(* Logix 5000 project; controller QW361 vendor 1 type 14 code 107 rev 32.11; software revision 32.00; part 14 of 20 *)

        [1996].log_data[0].time := 300.0, [1996].log_data[0].minminute := 50, [1996].log_data[0].maxminute := 50, [1996].log_data[0].valid := 1, [1996].log_data[1].valid := 1, [1996].log_data[2].valid := 1, [1996].log_data[3].valid := 1, [1996].log_data[4].valid := 1, [1996].time.Year := 2022, [1996].time.Month := 4, [1996].time.Day := 30, [1996].time.Hour := 19, [1996].time.Minute := 54, [1996].time.Second := 59, [1996].time.DST_ON := 1, [1997].log_data[0].min := 1.0, [1997].log_data[0].max := 1.0, [1997].log_data[0].total := 300.0, [1997].log_data[0].time := 300.0, [1997].log_data[0].minminute := 55, [1997].log_data[0].maxminute := 55, [1997].log_data[0].valid := 1, [1997].log_data[1].valid := 1, [1997].log_data[2].valid := 1, [1997].log_data[3].valid := 1, [1997].log_data[4].valid := 1, [1997].time.Year := 2022, [1997].time.Month := 4, [1997].time.Day := 30, [1997].time.Hour := 19, [1997].time.Minute := 59, [1997].time.Second := 59, [1997].time.DST_ON := 1, [1998].log_data[0].min := 1.0, [1998].log_data[0].max := 1.0, [1998].log_data[0].total := 300.0, [1998].log_data[0].time := 300.0, [1998].log_data[0].valid := 1, [1998].log_data[1].valid := 1, [1998].log_data[2].valid := 1, [1998].log_data[3].valid := 1, [1998].log_data[4].valid := 1, [1998].time.Year := 2022, [1998].time.Month := 4, [1998].time.Day := 30, [1998].time.Hour := 20, [1998].time.Minute := 4, [1998].time.Second := 59, [1998].time.DST_ON := 1, [1999].log_data[0].min := 1.0, [1999].log_data[0].max := 1.0, [1999].log_data[0].total := 300.0, [1999].log_data[0].time := 300.0, [1999].log_data[0].minminute := 5, [1999].log_data[0].maxminute := 5, [1999].log_data[0].valid := 1, [1999].log_data[1].valid := 1, [1999].log_data[2].valid := 1, [1999].log_data[3].valid := 1, [1999].log_data[4].valid := 1,
        [1999].time.Year := 2022, [1999].time.Month := 4, [1999].time.Day := 30, [1999].time.Hour := 20, [1999].time.Minute := 9, [1999].time.Second := 59, [1999].time.DST_ON := 1, [2000].log_data[0].min := 1.0, [2000].log_data[0].max := 1.0, [2000].log_data[0].total := 300.0, [2000].log_data[0].time := 300.0, [2000].log_data[0].minminute := 10, [2000].log_data[0].maxminute := 10, [2000].log_data[0].valid := 1, [2000].log_data[1].valid := 1, [2000].log_data[2].valid := 1, [2000].log_data[3].valid := 1, [2000].log_data[4].valid := 1, [2000].time.Year := 2022, [2000].time.Month := 4, [2000].time.Day := 30, [2000].time.Hour := 20, [2000].time.Minute := 14, [2000].time.Second := 59, [2000].time.DST_ON := 1, [2001].log_data[0].min := 1.0, [2001].log_data[0].max := 1.0, [2001].log_data[0].total := 300.0, [2001].log_data[0].time := 300.0, [2001].log_data[0].minminute := 15, [2001].log_data[0].maxminute := 15, [2001].log_data[0].valid := 1, [2001].log_data[1].valid := 1, [2001].log_data[2].valid := 1, [2001].log_data[3].valid := 1, [2001].log_data[4].valid := 1, [2001].time.Year := 2022, [2001].time.Month := 4, [2001].time.Day := 30, [2001].time.Hour := 20, [2001].time.Minute := 19, [2001].time.Second := 59, [2001].time.DST_ON := 1, [2002].log_data[0].min := 1.0, [2002].log_data[0].max := 1.0, [2002].log_data[0].total := 300.0, [2002].log_data[0].time := 300.0, [2002].log_data[0].minminute := 20, [2002].log_data[0].maxminute := 20, [2002].log_data[0].valid := 1, [2002].log_data[1].valid := 1, [2002].log_data[2].valid := 1, [2002].log_data[3].valid := 1, [2002].log_data[4].valid := 1, [2002].time.Year := 2022, [2002].time.Month := 4, [2002].time.Day := 30, [2002].time.Hour := 20, [2002].time.Minute := 24, [2002].time.Second := 59,
        [2002].time.DST_ON := 1, [2003].log_data[0].min := 1.0, [2003].log_data[0].max := 1.0, [2003].log_data[0].total := 300.0, [2003].log_data[0].time := 300.0, [2003].log_data[0].minminute := 25, [2003].log_data[0].maxminute := 25, [2003].log_data[0].valid := 1, [2003].log_data[1].valid := 1, [2003].log_data[2].valid := 1, [2003].log_data[3].valid := 1, [2003].log_data[4].valid := 1, [2003].time.Year := 2022, [2003].time.Month := 4, [2003].time.Day := 30, [2003].time.Hour := 20, [2003].time.Minute := 29, [2003].time.Second := 59, [2003].time.DST_ON := 1, [2004].log_data[0].min := 1.0, [2004].log_data[0].max := 1.0, [2004].log_data[0].total := 300.0, [2004].log_data[0].time := 300.0, [2004].log_data[0].minminute := 30, [2004].log_data[0].maxminute := 30, [2004].log_data[0].valid := 1, [2004].log_data[1].valid := 1, [2004].log_data[2].valid := 1, [2004].log_data[3].valid := 1, [2004].log_data[4].valid := 1, [2004].time.Year := 2022, [2004].time.Month := 4, [2004].time.Day := 30, [2004].time.Hour := 20, [2004].time.Minute := 34, [2004].time.Second := 59, [2004].time.DST_ON := 1, [2005].log_data[0].min := 1.0, [2005].log_data[0].max := 1.0, [2005].log_data[0].total := 300.0, [2005].log_data[0].time := 300.0, [2005].log_data[0].minminute := 35, [2005].log_data[0].maxminute := 35, [2005].log_data[0].valid := 1, [2005].log_data[1].valid := 1, [2005].log_data[2].valid := 1, [2005].log_data[3].valid := 1, [2005].log_data[4].valid := 1, [2005].time.Year := 2022, [2005].time.Month := 4, [2005].time.Day := 30, [2005].time.Hour := 20, [2005].time.Minute := 39, [2005].time.Second := 59, [2005].time.DST_ON := 1, [2006].log_data[0].min := 1.0, [2006].log_data[0].max := 1.0, [2006].log_data[0].total := 300.0, [2006].log_data[0].time := 300.0, [2006].log_data[0].minminute := 40,
        [2006].log_data[0].maxminute := 40, [2006].log_data[0].valid := 1, [2006].log_data[1].valid := 1, [2006].log_data[2].valid := 1, [2006].log_data[3].valid := 1, [2006].log_data[4].valid := 1, [2006].time.Year := 2022, [2006].time.Month := 4, [2006].time.Day := 30, [2006].time.Hour := 20, [2006].time.Minute := 44, [2006].time.Second := 59, [2006].time.DST_ON := 1, [2007].log_data[0].min := 1.0, [2007].log_data[0].max := 1.0, [2007].log_data[0].total := 300.0, [2007].log_data[0].time := 300.0, [2007].log_data[0].minminute := 45, [2007].log_data[0].maxminute := 45, [2007].log_data[0].valid := 1, [2007].log_data[1].valid := 1, [2007].log_data[2].valid := 1, [2007].log_data[3].valid := 1, [2007].log_data[4].valid := 1, [2007].time.Year := 2022, [2007].time.Month := 4, [2007].time.Day := 30, [2007].time.Hour := 20, [2007].time.Minute := 49, [2007].time.Second := 59, [2007].time.DST_ON := 1, [2008].log_data[0].min := 1.0, [2008].log_data[0].max := 1.0, [2008].log_data[0].total := 300.001, [2008].log_data[0].time := 300.001, [2008].log_data[0].minminute := 50, [2008].log_data[0].maxminute := 50, [2008].log_data[0].valid := 1, [2008].log_data[1].valid := 1, [2008].log_data[2].valid := 1, [2008].log_data[3].valid := 1, [2008].log_data[4].valid := 1, [2008].time.Year := 2022, [2008].time.Month := 4, [2008].time.Day := 30, [2008].time.Hour := 20, [2008].time.Minute := 54, [2008].time.Second := 59, [2008].time.DST_ON := 1, [2009].log_data[0].min := 1.0, [2009].log_data[0].max := 1.0, [2009].log_data[0].total := 300.001, [2009].log_data[0].time := 300.001, [2009].log_data[0].minminute := 55, [2009].log_data[0].maxminute := 55, [2009].log_data[0].valid := 1, [2009].log_data[1].valid := 1, [2009].log_data[2].valid := 1, [2009].log_data[3].valid := 1, [2009].log_data[4].valid := 1,
        [2009].time.Year := 2022, [2009].time.Month := 4, [2009].time.Day := 30, [2009].time.Hour := 20, [2009].time.Minute := 59, [2009].time.Second := 59, [2009].time.DST_ON := 1, [2010].log_data[0].min := 1.0, [2010].log_data[0].max := 1.0, [2010].log_data[0].total := 300.0, [2010].log_data[0].time := 300.0, [2010].log_data[0].valid := 1, [2010].log_data[1].valid := 1, [2010].log_data[2].valid := 1, [2010].log_data[3].valid := 1, [2010].log_data[4].valid := 1, [2010].time.Year := 2022, [2010].time.Month := 4, [2010].time.Day := 30, [2010].time.Hour := 21, [2010].time.Minute := 4, [2010].time.Second := 59, [2010].time.DST_ON := 1, [2011].log_data[0].min := 1.0, [2011].log_data[0].max := 1.0, [2011].log_data[0].total := 300.0, [2011].log_data[0].time := 300.0, [2011].log_data[0].minminute := 5, [2011].log_data[0].maxminute := 5, [2011].log_data[0].valid := 1, [2011].log_data[1].valid := 1, [2011].log_data[2].valid := 1, [2011].log_data[3].valid := 1, [2011].log_data[4].valid := 1, [2011].time.Year := 2022, [2011].time.Month := 4, [2011].time.Day := 30, [2011].time.Hour := 21, [2011].time.Minute := 9, [2011].time.Second := 59, [2011].time.DST_ON := 1, [2012].log_data[0].min := 1.0, [2012].log_data[0].max := 1.0, [2012].log_data[0].total := 300.0, [2012].log_data[0].time := 300.0, [2012].log_data[0].minminute := 10, [2012].log_data[0].maxminute := 10, [2012].log_data[0].valid := 1, [2012].log_data[1].valid := 1, [2012].log_data[2].valid := 1, [2012].log_data[3].valid := 1, [2012].log_data[4].valid := 1, [2012].time.Year := 2022, [2012].time.Month := 4, [2012].time.Day := 30, [2012].time.Hour := 21, [2012].time.Minute := 14, [2012].time.Second := 59, [2012].time.DST_ON := 1, [2013].log_data[0].min := 1.0,
        [2013].log_data[0].max := 1.0, [2013].log_data[0].total := 300.0, [2013].log_data[0].time := 300.0, [2013].log_data[0].minminute := 15, [2013].log_data[0].maxminute := 15, [2013].log_data[0].valid := 1, [2013].log_data[1].valid := 1, [2013].log_data[2].valid := 1, [2013].log_data[3].valid := 1, [2013].log_data[4].valid := 1, [2013].time.Year := 2022, [2013].time.Month := 4, [2013].time.Day := 30, [2013].time.Hour := 21, [2013].time.Minute := 19, [2013].time.Second := 59, [2013].time.DST_ON := 1, [2014].log_data[0].min := 1.0, [2014].log_data[0].max := 1.0, [2014].log_data[0].total := 300.0, [2014].log_data[0].time := 300.0, [2014].log_data[0].minminute := 20, [2014].log_data[0].maxminute := 20, [2014].log_data[0].valid := 1, [2014].log_data[1].valid := 1, [2014].log_data[2].valid := 1, [2014].log_data[3].valid := 1, [2014].log_data[4].valid := 1, [2014].time.Year := 2022, [2014].time.Month := 4, [2014].time.Day := 30, [2014].time.Hour := 21, [2014].time.Minute := 24, [2014].time.Second := 59, [2014].time.DST_ON := 1, [2015].log_data[0].min := 1.0, [2015].log_data[0].max := 1.0, [2015].log_data[0].total := 300.0, [2015].log_data[0].time := 300.0, [2015].log_data[0].minminute := 25, [2015].log_data[0].maxminute := 25, [2015].log_data[0].valid := 1, [2015].log_data[1].valid := 1, [2015].log_data[2].valid := 1, [2015].log_data[3].valid := 1, [2015].log_data[4].valid := 1, [2015].time.Year := 2022, [2015].time.Month := 4, [2015].time.Day := 30, [2015].time.Hour := 21, [2015].time.Minute := 29, [2015].time.Second := 59, [2015].time.DST_ON := 1, [2016].log_data[0].min := 1.0, [2016].log_data[0].max := 1.0, [2016].log_data[0].total := 300.0, [2016].log_data[0].time := 300.0, [2016].log_data[0].minminute := 30, [2016].log_data[0].maxminute := 30, [2016].log_data[0].valid := 1,
        [2016].log_data[1].valid := 1, [2016].log_data[2].valid := 1, [2016].log_data[3].valid := 1, [2016].log_data[4].valid := 1, [2016].time.Year := 2022, [2016].time.Month := 4, [2016].time.Day := 30, [2016].time.Hour := 21, [2016].time.Minute := 34, [2016].time.Second := 59, [2016].time.DST_ON := 1, [2017].log_data[0].min := 1.0, [2017].log_data[0].max := 1.0, [2017].log_data[0].total := 300.0, [2017].log_data[0].time := 300.0, [2017].log_data[0].minminute := 35, [2017].log_data[0].maxminute := 35, [2017].log_data[0].valid := 1, [2017].log_data[1].valid := 1, [2017].log_data[2].valid := 1, [2017].log_data[3].valid := 1, [2017].log_data[4].valid := 1, [2017].time.Year := 2022, [2017].time.Month := 4, [2017].time.Day := 30, [2017].time.Hour := 21, [2017].time.Minute := 39, [2017].time.Second := 59, [2017].time.DST_ON := 1, [2018].log_data[0].min := 1.0, [2018].log_data[0].max := 1.0, [2018].log_data[0].total := 300.0, [2018].log_data[0].time := 300.0, [2018].log_data[0].minminute := 40, [2018].log_data[0].maxminute := 40, [2018].log_data[0].valid := 1, [2018].log_data[1].valid := 1, [2018].log_data[2].valid := 1, [2018].log_data[3].valid := 1, [2018].log_data[4].valid := 1, [2018].time.Year := 2022, [2018].time.Month := 4, [2018].time.Day := 30, [2018].time.Hour := 21, [2018].time.Minute := 44, [2018].time.Second := 59, [2018].time.DST_ON := 1, [2019].log_data[0].min := 1.0, [2019].log_data[0].max := 1.0, [2019].log_data[0].total := 300.0, [2019].log_data[0].time := 300.0, [2019].log_data[0].minminute := 45, [2019].log_data[0].maxminute := 45, [2019].log_data[0].valid := 1, [2019].log_data[1].valid := 1, [2019].log_data[2].valid := 1, [2019].log_data[3].valid := 1, [2019].log_data[4].valid := 1, [2019].time.Year := 2022, [2019].time.Month := 4,
        [2019].time.Day := 30, [2019].time.Hour := 21, [2019].time.Minute := 49, [2019].time.Second := 59, [2019].time.DST_ON := 1, [2020].log_data[0].min := 1.0, [2020].log_data[0].max := 1.0, [2020].log_data[0].total := 300.0, [2020].log_data[0].time := 300.0, [2020].log_data[0].minminute := 50, [2020].log_data[0].maxminute := 50, [2020].log_data[0].valid := 1, [2020].log_data[1].valid := 1, [2020].log_data[2].valid := 1, [2020].log_data[3].valid := 1, [2020].log_data[4].valid := 1, [2020].time.Year := 2022, [2020].time.Month := 4, [2020].time.Day := 30, [2020].time.Hour := 21, [2020].time.Minute := 54, [2020].time.Second := 59, [2020].time.DST_ON := 1, [2021].log_data[0].min := 1.0, [2021].log_data[0].max := 1.0, [2021].log_data[0].total := 300.0, [2021].log_data[0].time := 300.0, [2021].log_data[0].minminute := 55, [2021].log_data[0].maxminute := 55, [2021].log_data[0].valid := 1, [2021].log_data[1].valid := 1, [2021].log_data[2].valid := 1, [2021].log_data[3].valid := 1, [2021].log_data[4].valid := 1, [2021].time.Year := 2022, [2021].time.Month := 4, [2021].time.Day := 30, [2021].time.Hour := 21, [2021].time.Minute := 59, [2021].time.Second := 59, [2021].time.DST_ON := 1, [2022].log_data[0].min := 1.0, [2022].log_data[0].max := 1.0, [2022].log_data[0].total := 300.0, [2022].log_data[0].time := 300.0, [2022].log_data[0].valid := 1, [2022].log_data[1].valid := 1, [2022].log_data[2].valid := 1, [2022].log_data[3].valid := 1, [2022].log_data[4].valid := 1, [2022].time.Year := 2022, [2022].time.Month := 4, [2022].time.Day := 30, [2022].time.Hour := 22, [2022].time.Minute := 4, [2022].time.Second := 59, [2022].time.DST_ON := 1, [2023].log_data[0].min := 1.0, [2023].log_data[0].max := 1.0, [2023].log_data[0].total := 300.0,
        [2023].log_data[0].time := 300.0, [2023].log_data[0].minminute := 5, [2023].log_data[0].maxminute := 5, [2023].log_data[0].valid := 1, [2023].log_data[1].valid := 1, [2023].log_data[2].valid := 1, [2023].log_data[3].valid := 1, [2023].log_data[4].valid := 1, [2023].time.Year := 2022, [2023].time.Month := 4, [2023].time.Day := 30, [2023].time.Hour := 22, [2023].time.Minute := 9, [2023].time.Second := 59, [2023].time.DST_ON := 1, [2024].log_data[0].min := 1.0, [2024].log_data[0].max := 1.0, [2024].log_data[0].total := 300.0, [2024].log_data[0].time := 300.0, [2024].log_data[0].minminute := 10, [2024].log_data[0].maxminute := 10, [2024].log_data[0].valid := 1, [2024].log_data[1].valid := 1, [2024].log_data[2].valid := 1, [2024].log_data[3].valid := 1, [2024].log_data[4].valid := 1, [2024].time.Year := 2022, [2024].time.Month := 4, [2024].time.Day := 30, [2024].time.Hour := 22, [2024].time.Minute := 14, [2024].time.Second := 59, [2024].time.DST_ON := 1, [2025].log_data[0].min := 1.0, [2025].log_data[0].max := 1.0, [2025].log_data[0].total := 300.0, [2025].log_data[0].time := 300.0, [2025].log_data[0].minminute := 15, [2025].log_data[0].maxminute := 15, [2025].log_data[0].valid := 1, [2025].log_data[1].valid := 1, [2025].log_data[2].valid := 1, [2025].log_data[3].valid := 1, [2025].log_data[4].valid := 1, [2025].time.Year := 2022, [2025].time.Month := 4, [2025].time.Day := 30, [2025].time.Hour := 22, [2025].time.Minute := 19, [2025].time.Second := 59, [2025].time.DST_ON := 1, [2026].log_data[0].min := 1.0, [2026].log_data[0].max := 1.0, [2026].log_data[0].total := 300.0, [2026].log_data[0].time := 300.0, [2026].log_data[0].minminute := 20, [2026].log_data[0].maxminute := 20, [2026].log_data[0].valid := 1, [2026].log_data[1].valid := 1, [2026].log_data[2].valid := 1,
        [2026].log_data[3].valid := 1, [2026].log_data[4].valid := 1, [2026].time.Year := 2022, [2026].time.Month := 4, [2026].time.Day := 30, [2026].time.Hour := 22, [2026].time.Minute := 24, [2026].time.Second := 59, [2026].time.DST_ON := 1, [2027].log_data[0].min := 1.0, [2027].log_data[0].max := 1.0, [2027].log_data[0].total := 300.0, [2027].log_data[0].time := 300.0, [2027].log_data[0].minminute := 25, [2027].log_data[0].maxminute := 25, [2027].log_data[0].valid := 1, [2027].log_data[1].valid := 1, [2027].log_data[2].valid := 1, [2027].log_data[3].valid := 1, [2027].log_data[4].valid := 1, [2027].time.Year := 2022, [2027].time.Month := 4, [2027].time.Day := 30, [2027].time.Hour := 22, [2027].time.Minute := 29, [2027].time.Second := 59, [2027].time.DST_ON := 1, [2028].log_data[0].min := 1.0, [2028].log_data[0].max := 1.0, [2028].log_data[0].total := 300.0, [2028].log_data[0].time := 300.0, [2028].log_data[0].minminute := 30, [2028].log_data[0].maxminute := 30, [2028].log_data[0].valid := 1, [2028].log_data[1].valid := 1, [2028].log_data[2].valid := 1, [2028].log_data[3].valid := 1, [2028].log_data[4].valid := 1, [2028].time.Year := 2022, [2028].time.Month := 4, [2028].time.Day := 30, [2028].time.Hour := 22, [2028].time.Minute := 34, [2028].time.Second := 59, [2028].time.DST_ON := 1, [2029].log_data[0].min := 1.0, [2029].log_data[0].max := 1.0, [2029].log_data[0].total := 300.0, [2029].log_data[0].time := 300.0, [2029].log_data[0].minminute := 35, [2029].log_data[0].maxminute := 35, [2029].log_data[0].valid := 1, [2029].log_data[1].valid := 1, [2029].log_data[2].valid := 1, [2029].log_data[3].valid := 1, [2029].log_data[4].valid := 1, [2029].time.Year := 2022, [2029].time.Month := 4, [2029].time.Day := 30, [2029].time.Hour := 22,
        [2029].time.Minute := 39, [2029].time.Second := 59, [2029].time.DST_ON := 1, [2030].log_data[0].min := 1.0, [2030].log_data[0].max := 1.0, [2030].log_data[0].total := 300.0, [2030].log_data[0].time := 300.0, [2030].log_data[0].minminute := 40, [2030].log_data[0].maxminute := 40, [2030].log_data[0].valid := 1, [2030].log_data[1].valid := 1, [2030].log_data[2].valid := 1, [2030].log_data[3].valid := 1, [2030].log_data[4].valid := 1, [2030].time.Year := 2022, [2030].time.Month := 4, [2030].time.Day := 30, [2030].time.Hour := 22, [2030].time.Minute := 44, [2030].time.Second := 59, [2030].time.DST_ON := 1, [2031].log_data[0].min := 1.0, [2031].log_data[0].max := 1.0, [2031].log_data[0].total := 300.0, [2031].log_data[0].time := 300.0, [2031].log_data[0].minminute := 45, [2031].log_data[0].maxminute := 45, [2031].log_data[0].valid := 1, [2031].log_data[1].valid := 1, [2031].log_data[2].valid := 1, [2031].log_data[3].valid := 1, [2031].log_data[4].valid := 1, [2031].time.Year := 2022, [2031].time.Month := 4, [2031].time.Day := 30, [2031].time.Hour := 22, [2031].time.Minute := 49, [2031].time.Second := 59, [2031].time.DST_ON := 1, [2032].log_data[0].min := 1.0, [2032].log_data[0].max := 1.0, [2032].log_data[0].total := 300.0, [2032].log_data[0].time := 300.0, [2032].log_data[0].minminute := 50, [2032].log_data[0].maxminute := 50, [2032].log_data[0].valid := 1, [2032].log_data[1].valid := 1, [2032].log_data[2].valid := 1, [2032].log_data[3].valid := 1, [2032].log_data[4].valid := 1, [2032].time.Year := 2022, [2032].time.Month := 4, [2032].time.Day := 30, [2032].time.Hour := 22, [2032].time.Minute := 54, [2032].time.Second := 59, [2032].time.DST_ON := 1, [2033].log_data[0].min := 1.0, [2033].log_data[0].max := 1.0, [2033].log_data[0].total := 300.0,
        [2033].log_data[0].time := 300.0, [2033].log_data[0].minminute := 55, [2033].log_data[0].maxminute := 55, [2033].log_data[0].valid := 1, [2033].log_data[1].valid := 1, [2033].log_data[2].valid := 1, [2033].log_data[3].valid := 1, [2033].log_data[4].valid := 1, [2033].time.Year := 2022, [2033].time.Month := 4, [2033].time.Day := 30, [2033].time.Hour := 22, [2033].time.Minute := 59, [2033].time.Second := 59, [2033].time.DST_ON := 1, [2034].log_data[0].min := 1.0, [2034].log_data[0].max := 1.0, [2034].log_data[0].total := 300.0, [2034].log_data[0].time := 300.0, [2034].log_data[0].valid := 1, [2034].log_data[1].valid := 1, [2034].log_data[2].valid := 1, [2034].log_data[3].valid := 1, [2034].log_data[4].valid := 1, [2034].time.Year := 2022, [2034].time.Month := 4, [2034].time.Day := 30, [2034].time.Hour := 23, [2034].time.Minute := 4, [2034].time.Second := 59, [2034].time.DST_ON := 1, [2035].log_data[0].min := 1.0, [2035].log_data[0].max := 1.0, [2035].log_data[0].total := 300.0, [2035].log_data[0].time := 300.0, [2035].log_data[0].minminute := 5, [2035].log_data[0].maxminute := 5, [2035].log_data[0].valid := 1, [2035].log_data[1].valid := 1, [2035].log_data[2].valid := 1, [2035].log_data[3].valid := 1, [2035].log_data[4].valid := 1, [2035].time.Year := 2022, [2035].time.Month := 4, [2035].time.Day := 30, [2035].time.Hour := 23, [2035].time.Minute := 9, [2035].time.Second := 59, [2035].time.DST_ON := 1, [2036].log_data[0].min := 1.0, [2036].log_data[0].max := 1.0, [2036].log_data[0].total := 300.0, [2036].log_data[0].time := 300.0, [2036].log_data[0].minminute := 10, [2036].log_data[0].maxminute := 10, [2036].log_data[0].valid := 1, [2036].log_data[1].valid := 1, [2036].log_data[2].valid := 1, [2036].log_data[3].valid := 1, [2036].log_data[4].valid := 1,
        [2036].time.Year := 2022, [2036].time.Month := 4, [2036].time.Day := 30, [2036].time.Hour := 23, [2036].time.Minute := 14, [2036].time.Second := 59, [2036].time.DST_ON := 1, [2037].log_data[0].min := 1.0, [2037].log_data[0].max := 1.0, [2037].log_data[0].total := 300.0, [2037].log_data[0].time := 300.0, [2037].log_data[0].minminute := 15, [2037].log_data[0].maxminute := 15, [2037].log_data[0].valid := 1, [2037].log_data[1].valid := 1, [2037].log_data[2].valid := 1, [2037].log_data[3].valid := 1, [2037].log_data[4].valid := 1, [2037].time.Year := 2022, [2037].time.Month := 4, [2037].time.Day := 30, [2037].time.Hour := 23, [2037].time.Minute := 19, [2037].time.Second := 59, [2037].time.DST_ON := 1, [2038].log_data[0].min := 1.0, [2038].log_data[0].max := 1.0, [2038].log_data[0].total := 300.0, [2038].log_data[0].time := 300.0, [2038].log_data[0].minminute := 20, [2038].log_data[0].maxminute := 20, [2038].log_data[0].valid := 1, [2038].log_data[1].valid := 1, [2038].log_data[2].valid := 1, [2038].log_data[3].valid := 1, [2038].log_data[4].valid := 1, [2038].time.Year := 2022, [2038].time.Month := 4, [2038].time.Day := 30, [2038].time.Hour := 23, [2038].time.Minute := 24, [2038].time.Second := 59, [2038].time.DST_ON := 1, [2039].log_data[0].min := 1.0, [2039].log_data[0].max := 1.0, [2039].log_data[0].total := 300.0, [2039].log_data[0].time := 300.0, [2039].log_data[0].minminute := 25, [2039].log_data[0].maxminute := 25, [2039].log_data[0].valid := 1, [2039].log_data[1].valid := 1, [2039].log_data[2].valid := 1, [2039].log_data[3].valid := 1, [2039].log_data[4].valid := 1, [2039].time.Year := 2022, [2039].time.Month := 4, [2039].time.Day := 30, [2039].time.Hour := 23, [2039].time.Minute := 29, [2039].time.Second := 59,
        [2039].time.DST_ON := 1, [2040].log_data[0].min := 1.0, [2040].log_data[0].max := 1.0, [2040].log_data[0].total := 300.0, [2040].log_data[0].time := 300.0, [2040].log_data[0].minminute := 30, [2040].log_data[0].maxminute := 30, [2040].log_data[0].valid := 1, [2040].log_data[1].valid := 1, [2040].log_data[2].valid := 1, [2040].log_data[3].valid := 1, [2040].log_data[4].valid := 1, [2040].time.Year := 2022, [2040].time.Month := 4, [2040].time.Day := 30, [2040].time.Hour := 23, [2040].time.Minute := 34, [2040].time.Second := 59, [2040].time.DST_ON := 1, [2041].log_data[0].min := 1.0, [2041].log_data[0].max := 1.0, [2041].log_data[0].total := 300.0, [2041].log_data[0].time := 300.0, [2041].log_data[0].minminute := 35, [2041].log_data[0].maxminute := 35, [2041].log_data[0].valid := 1, [2041].log_data[1].valid := 1, [2041].log_data[2].valid := 1, [2041].log_data[3].valid := 1, [2041].log_data[4].valid := 1, [2041].time.Year := 2022, [2041].time.Month := 4, [2041].time.Day := 30, [2041].time.Hour := 23, [2041].time.Minute := 39, [2041].time.Second := 59, [2041].time.DST_ON := 1, [2042].log_data[0].min := 1.0, [2042].log_data[0].max := 1.0, [2042].log_data[0].total := 300.0, [2042].log_data[0].time := 300.0, [2042].log_data[0].minminute := 40, [2042].log_data[0].maxminute := 40, [2042].log_data[0].valid := 1, [2042].log_data[1].valid := 1, [2042].log_data[2].valid := 1, [2042].log_data[3].valid := 1, [2042].log_data[4].valid := 1, [2042].time.Year := 2022, [2042].time.Month := 4, [2042].time.Day := 30, [2042].time.Hour := 23, [2042].time.Minute := 44, [2042].time.Second := 59, [2042].time.DST_ON := 1, [2043].log_data[0].min := 1.0, [2043].log_data[0].max := 1.0, [2043].log_data[0].total := 300.0, [2043].log_data[0].time := 300.0, [2043].log_data[0].minminute := 45,
        [2043].log_data[0].maxminute := 45, [2043].log_data[0].valid := 1, [2043].log_data[1].valid := 1, [2043].log_data[2].valid := 1, [2043].log_data[3].valid := 1, [2043].log_data[4].valid := 1, [2043].time.Year := 2022, [2043].time.Month := 4, [2043].time.Day := 30, [2043].time.Hour := 23, [2043].time.Minute := 49, [2043].time.Second := 59, [2043].time.DST_ON := 1, [2044].log_data[0].min := 1.0, [2044].log_data[0].max := 1.0, [2044].log_data[0].total := 300.0, [2044].log_data[0].time := 300.0, [2044].log_data[0].minminute := 50, [2044].log_data[0].maxminute := 50, [2044].log_data[0].valid := 1, [2044].log_data[1].valid := 1, [2044].log_data[2].valid := 1, [2044].log_data[3].valid := 1, [2044].log_data[4].valid := 1, [2044].time.Year := 2022, [2044].time.Month := 4, [2044].time.Day := 30, [2044].time.Hour := 23, [2044].time.Minute := 54, [2044].time.Second := 59, [2044].time.DST_ON := 1, [2045].log_data[0].min := 1.0, [2045].log_data[0].max := 1.0, [2045].log_data[0].total := 300.0, [2045].log_data[0].time := 300.0, [2045].log_data[0].minminute := 55, [2045].log_data[0].maxminute := 55, [2045].log_data[0].valid := 1, [2045].log_data[1].valid := 1, [2045].log_data[2].valid := 1, [2045].log_data[3].valid := 1, [2045].log_data[4].valid := 1, [2045].time.Year := 2022, [2045].time.Month := 4, [2045].time.Day := 30, [2045].time.Hour := 23, [2045].time.Minute := 59, [2045].time.Second := 59, [2045].time.DST_ON := 1, [2046].log_data[0].min := 1.0, [2046].log_data[0].max := 1.0, [2046].log_data[0].total := 300.0, [2046].log_data[0].time := 300.0, [2046].log_data[0].valid := 1, [2046].log_data[1].valid := 1, [2046].log_data[2].valid := 1, [2046].log_data[3].valid := 1, [2046].log_data[4].valid := 1, [2046].time.Year := 2022, [2046].time.Month := 5,
        [2046].time.Day := 1, [2046].time.Minute := 4, [2046].time.Second := 59, [2046].time.DST_ON := 1, [2047].log_data[0].min := 1.0, [2047].log_data[0].max := 1.0, [2047].log_data[0].total := 300.0, [2047].log_data[0].time := 300.0, [2047].log_data[0].minminute := 5, [2047].log_data[0].maxminute := 5, [2047].log_data[0].valid := 1, [2047].log_data[1].valid := 1, [2047].log_data[2].valid := 1, [2047].log_data[3].valid := 1, [2047].log_data[4].valid := 1, [2047].time.Year := 2022, [2047].time.Month := 5, [2047].time.Day := 1, [2047].time.Minute := 9, [2047].time.Second := 59, [2047].time.DST_ON := 1, [2048].log_data[0].min := 1.0, [2048].log_data[0].max := 1.0, [2048].log_data[0].total := 300.0, [2048].log_data[0].time := 300.0, [2048].log_data[0].minminute := 10, [2048].log_data[0].maxminute := 10, [2048].log_data[0].valid := 1, [2048].log_data[1].valid := 1, [2048].log_data[2].valid := 1, [2048].log_data[3].valid := 1, [2048].log_data[4].valid := 1, [2048].time.Year := 2022, [2048].time.Month := 5, [2048].time.Day := 1, [2048].time.Minute := 14, [2048].time.Second := 59, [2048].time.DST_ON := 1, [2049].log_data[0].min := 1.0, [2049].log_data[0].max := 1.0, [2049].log_data[0].total := 300.0, [2049].log_data[0].time := 300.0, [2049].log_data[0].minminute := 15, [2049].log_data[0].maxminute := 15, [2049].log_data[0].valid := 1, [2049].log_data[1].valid := 1, [2049].log_data[2].valid := 1, [2049].log_data[3].valid := 1, [2049].log_data[4].valid := 1, [2049].time.Year := 2022, [2049].time.Month := 5, [2049].time.Day := 1, [2049].time.Minute := 19, [2049].time.Second := 59, [2049].time.DST_ON := 1, [2050].log_data[0].min := 1.0, [2050].log_data[0].max := 1.0, [2050].log_data[0].total := 300.0, [2050].log_data[0].time := 300.0, [2050].log_data[0].minminute := 20,
        [2050].log_data[0].maxminute := 20, [2050].log_data[0].valid := 1, [2050].log_data[1].valid := 1, [2050].log_data[2].valid := 1, [2050].log_data[3].valid := 1, [2050].log_data[4].valid := 1, [2050].time.Year := 2022, [2050].time.Month := 5, [2050].time.Day := 1, [2050].time.Minute := 24, [2050].time.Second := 59, [2050].time.DST_ON := 1, [2051].log_data[0].min := 1.0, [2051].log_data[0].max := 1.0, [2051].log_data[0].total := 300.0, [2051].log_data[0].time := 300.0, [2051].log_data[0].minminute := 25, [2051].log_data[0].maxminute := 25, [2051].log_data[0].valid := 1, [2051].log_data[1].valid := 1, [2051].log_data[2].valid := 1, [2051].log_data[3].valid := 1, [2051].log_data[4].valid := 1, [2051].time.Year := 2022, [2051].time.Month := 5, [2051].time.Day := 1, [2051].time.Minute := 29, [2051].time.Second := 59, [2051].time.DST_ON := 1, [2052].log_data[0].min := 1.0, [2052].log_data[0].max := 1.0, [2052].log_data[0].total := 300.0, [2052].log_data[0].time := 300.0, [2052].log_data[0].minminute := 30, [2052].log_data[0].maxminute := 30, [2052].log_data[0].valid := 1, [2052].log_data[1].valid := 1, [2052].log_data[2].valid := 1, [2052].log_data[3].valid := 1, [2052].log_data[4].valid := 1, [2052].time.Year := 2022, [2052].time.Month := 5, [2052].time.Day := 1, [2052].time.Minute := 34, [2052].time.Second := 59, [2052].time.DST_ON := 1, [2053].log_data[0].min := 1.0, [2053].log_data[0].max := 1.0, [2053].log_data[0].total := 299.999, [2053].log_data[0].time := 299.999, [2053].log_data[0].minminute := 35, [2053].log_data[0].maxminute := 35, [2053].log_data[0].valid := 1, [2053].log_data[1].valid := 1, [2053].log_data[2].valid := 1, [2053].log_data[3].valid := 1, [2053].log_data[4].valid := 1, [2053].time.Year := 2022, [2053].time.Month := 5, [2053].time.Day := 1,
        [2053].time.Minute := 39, [2053].time.Second := 59, [2053].time.DST_ON := 1, [2054].log_data[0].min := 1.0, [2054].log_data[0].max := 1.0, [2054].log_data[0].total := 300.0, [2054].log_data[0].time := 300.0, [2054].log_data[0].minminute := 40, [2054].log_data[0].maxminute := 40, [2054].log_data[0].valid := 1, [2054].log_data[1].valid := 1, [2054].log_data[2].valid := 1, [2054].log_data[3].valid := 1, [2054].log_data[4].valid := 1, [2054].time.Year := 2022, [2054].time.Month := 5, [2054].time.Day := 1, [2054].time.Minute := 44, [2054].time.Second := 59, [2054].time.DST_ON := 1, [2055].log_data[0].min := 1.0, [2055].log_data[0].max := 1.0, [2055].log_data[0].total := 300.0, [2055].log_data[0].time := 300.0, [2055].log_data[0].minminute := 45, [2055].log_data[0].maxminute := 45, [2055].log_data[0].valid := 1, [2055].log_data[1].valid := 1, [2055].log_data[2].valid := 1, [2055].log_data[3].valid := 1, [2055].log_data[4].valid := 1, [2055].time.Year := 2022, [2055].time.Month := 5, [2055].time.Day := 1, [2055].time.Minute := 49, [2055].time.Second := 59, [2055].time.DST_ON := 1, [2056].log_data[0].min := 1.0, [2056].log_data[0].max := 1.0, [2056].log_data[0].total := 300.0, [2056].log_data[0].time := 300.0, [2056].log_data[0].minminute := 50, [2056].log_data[0].maxminute := 50, [2056].log_data[0].valid := 1, [2056].log_data[1].valid := 1, [2056].log_data[2].valid := 1, [2056].log_data[3].valid := 1, [2056].log_data[4].valid := 1, [2056].time.Year := 2022, [2056].time.Month := 5, [2056].time.Day := 1, [2056].time.Minute := 54, [2056].time.Second := 59, [2056].time.DST_ON := 1, [2057].log_data[0].min := 1.0, [2057].log_data[0].max := 1.0, [2057].log_data[0].total := 300.001, [2057].log_data[0].time := 300.001, [2057].log_data[0].minminute := 55, [2057].log_data[0].maxminute := 55,
        [2057].log_data[0].valid := 1, [2057].log_data[1].valid := 1, [2057].log_data[2].valid := 1, [2057].log_data[3].valid := 1, [2057].log_data[4].valid := 1, [2057].time.Year := 2022, [2057].time.Month := 5, [2057].time.Day := 1, [2057].time.Minute := 59, [2057].time.Second := 59, [2057].time.DST_ON := 1, [2058].log_data[0].min := 1.0, [2058].log_data[0].max := 1.0, [2058].log_data[0].total := 300.0, [2058].log_data[0].time := 300.0, [2058].log_data[0].valid := 1, [2058].log_data[1].valid := 1, [2058].log_data[2].valid := 1, [2058].log_data[3].valid := 1, [2058].log_data[4].valid := 1, [2058].time.Year := 2022, [2058].time.Month := 5, [2058].time.Day := 1, [2058].time.Hour := 1, [2058].time.Minute := 4, [2058].time.Second := 59, [2058].time.DST_ON := 1, [2059].log_data[0].min := 1.0, [2059].log_data[0].max := 1.0, [2059].log_data[0].total := 300.0, [2059].log_data[0].time := 300.0, [2059].log_data[0].minminute := 5, [2059].log_data[0].maxminute := 5, [2059].log_data[0].valid := 1, [2059].log_data[1].valid := 1, [2059].log_data[2].valid := 1, [2059].log_data[3].valid := 1, [2059].log_data[4].valid := 1, [2059].time.Year := 2022, [2059].time.Month := 5, [2059].time.Day := 1, [2059].time.Hour := 1, [2059].time.Minute := 9, [2059].time.Second := 59, [2059].time.DST_ON := 1, [2060].log_data[0].min := 1.0, [2060].log_data[0].max := 1.0, [2060].log_data[0].total := 300.0, [2060].log_data[0].time := 300.0, [2060].log_data[0].minminute := 10, [2060].log_data[0].maxminute := 10, [2060].log_data[0].valid := 1, [2060].log_data[1].valid := 1, [2060].log_data[2].valid := 1, [2060].log_data[3].valid := 1, [2060].log_data[4].valid := 1, [2060].time.Year := 2022, [2060].time.Month := 5, [2060].time.Day := 1, [2060].time.Hour := 1,
        [2060].time.Minute := 14, [2060].time.Second := 59, [2060].time.DST_ON := 1, [2061].log_data[0].min := 1.0, [2061].log_data[0].max := 1.0, [2061].log_data[0].total := 300.0, [2061].log_data[0].time := 300.0, [2061].log_data[0].minminute := 15, [2061].log_data[0].maxminute := 15, [2061].log_data[0].valid := 1, [2061].log_data[1].valid := 1, [2061].log_data[2].valid := 1, [2061].log_data[3].valid := 1, [2061].log_data[4].valid := 1, [2061].time.Year := 2022, [2061].time.Month := 5, [2061].time.Day := 1, [2061].time.Hour := 1, [2061].time.Minute := 19, [2061].time.Second := 59, [2061].time.DST_ON := 1, [2062].log_data[0].min := 1.0, [2062].log_data[0].max := 1.0, [2062].log_data[0].total := 300.0, [2062].log_data[0].time := 300.0, [2062].log_data[0].minminute := 20, [2062].log_data[0].maxminute := 20, [2062].log_data[0].valid := 1, [2062].log_data[1].valid := 1, [2062].log_data[2].valid := 1, [2062].log_data[3].valid := 1, [2062].log_data[4].valid := 1, [2062].time.Year := 2022, [2062].time.Month := 5, [2062].time.Day := 1, [2062].time.Hour := 1, [2062].time.Minute := 24, [2062].time.Second := 59, [2062].time.DST_ON := 1, [2063].log_data[0].min := 1.0, [2063].log_data[0].max := 1.0, [2063].log_data[0].total := 300.0, [2063].log_data[0].time := 300.0, [2063].log_data[0].minminute := 25, [2063].log_data[0].maxminute := 25, [2063].log_data[0].valid := 1, [2063].log_data[1].valid := 1, [2063].log_data[2].valid := 1, [2063].log_data[3].valid := 1, [2063].log_data[4].valid := 1, [2063].time.Year := 2022, [2063].time.Month := 5, [2063].time.Day := 1, [2063].time.Hour := 1, [2063].time.Minute := 29, [2063].time.Second := 59, [2063].time.DST_ON := 1, [2064].log_data[0].min := 1.0, [2064].log_data[0].max := 1.0, [2064].log_data[0].total := 300.0,
        [2064].log_data[0].time := 300.0, [2064].log_data[0].minminute := 30, [2064].log_data[0].maxminute := 30, [2064].log_data[0].valid := 1, [2064].log_data[1].valid := 1, [2064].log_data[2].valid := 1, [2064].log_data[3].valid := 1, [2064].log_data[4].valid := 1, [2064].time.Year := 2022, [2064].time.Month := 5, [2064].time.Day := 1, [2064].time.Hour := 1, [2064].time.Minute := 34, [2064].time.Second := 59, [2064].time.DST_ON := 1, [2065].log_data[0].min := 1.0, [2065].log_data[0].max := 1.0, [2065].log_data[0].total := 300.0, [2065].log_data[0].time := 300.0, [2065].log_data[0].minminute := 35, [2065].log_data[0].maxminute := 35, [2065].log_data[0].valid := 1, [2065].log_data[1].valid := 1, [2065].log_data[2].valid := 1, [2065].log_data[3].valid := 1, [2065].log_data[4].valid := 1, [2065].time.Year := 2022, [2065].time.Month := 5, [2065].time.Day := 1, [2065].time.Hour := 1, [2065].time.Minute := 39, [2065].time.Second := 59, [2065].time.DST_ON := 1, [2066].log_data[0].min := 1.0, [2066].log_data[0].max := 1.0, [2066].log_data[0].total := 300.0, [2066].log_data[0].time := 300.0, [2066].log_data[0].minminute := 40, [2066].log_data[0].maxminute := 40, [2066].log_data[0].valid := 1, [2066].log_data[1].valid := 1, [2066].log_data[2].valid := 1, [2066].log_data[3].valid := 1, [2066].log_data[4].valid := 1, [2066].time.Year := 2022, [2066].time.Month := 5, [2066].time.Day := 1, [2066].time.Hour := 1, [2066].time.Minute := 44, [2066].time.Second := 59, [2066].time.DST_ON := 1, [2067].log_data[0].min := 1.0, [2067].log_data[0].max := 1.0, [2067].log_data[0].total := 300.0, [2067].log_data[0].time := 300.0, [2067].log_data[0].minminute := 45, [2067].log_data[0].maxminute := 45, [2067].log_data[0].valid := 1, [2067].log_data[1].valid := 1, [2067].log_data[2].valid := 1,
        [2067].log_data[3].valid := 1, [2067].log_data[4].valid := 1, [2067].time.Year := 2022, [2067].time.Month := 5, [2067].time.Day := 1, [2067].time.Hour := 1, [2067].time.Minute := 49, [2067].time.Second := 59, [2067].time.DST_ON := 1, [2068].log_data[0].min := 1.0, [2068].log_data[0].max := 1.0, [2068].log_data[0].total := 300.0, [2068].log_data[0].time := 300.0, [2068].log_data[0].minminute := 50, [2068].log_data[0].maxminute := 50, [2068].log_data[0].valid := 1, [2068].log_data[1].valid := 1, [2068].log_data[2].valid := 1, [2068].log_data[3].valid := 1, [2068].log_data[4].valid := 1, [2068].time.Year := 2022, [2068].time.Month := 5, [2068].time.Day := 1, [2068].time.Hour := 1, [2068].time.Minute := 54, [2068].time.Second := 59, [2068].time.DST_ON := 1, [2069].log_data[0].min := 1.0, [2069].log_data[0].max := 1.0, [2069].log_data[0].total := 300.0, [2069].log_data[0].time := 300.0, [2069].log_data[0].minminute := 55, [2069].log_data[0].maxminute := 55, [2069].log_data[0].valid := 1, [2069].log_data[1].valid := 1, [2069].log_data[2].valid := 1, [2069].log_data[3].valid := 1, [2069].log_data[4].valid := 1, [2069].time.Year := 2022, [2069].time.Month := 5, [2069].time.Day := 1, [2069].time.Hour := 1, [2069].time.Minute := 59, [2069].time.Second := 59, [2069].time.DST_ON := 1, [2070].log_data[0].min := 1.0, [2070].log_data[0].max := 1.0, [2070].log_data[0].total := 300.0, [2070].log_data[0].time := 300.0, [2070].log_data[0].valid := 1, [2070].log_data[1].valid := 1, [2070].log_data[2].valid := 1, [2070].log_data[3].valid := 1, [2070].log_data[4].valid := 1, [2070].time.Year := 2022, [2070].time.Month := 5, [2070].time.Day := 1, [2070].time.Hour := 2, [2070].time.Minute := 4, [2070].time.Second := 59,
        [2070].time.DST_ON := 1, [2071].log_data[0].min := 1.0, [2071].log_data[0].max := 1.0, [2071].log_data[0].total := 300.0, [2071].log_data[0].time := 300.0, [2071].log_data[0].minminute := 5, [2071].log_data[0].maxminute := 5, [2071].log_data[0].valid := 1, [2071].log_data[1].valid := 1, [2071].log_data[2].valid := 1, [2071].log_data[3].valid := 1, [2071].log_data[4].valid := 1, [2071].time.Year := 2022, [2071].time.Month := 5, [2071].time.Day := 1, [2071].time.Hour := 2, [2071].time.Minute := 9, [2071].time.Second := 59, [2071].time.DST_ON := 1, [2072].log_data[0].min := 1.0, [2072].log_data[0].max := 1.0, [2072].log_data[0].total := 300.0, [2072].log_data[0].time := 300.0, [2072].log_data[0].minminute := 10, [2072].log_data[0].maxminute := 10, [2072].log_data[0].valid := 1, [2072].log_data[1].valid := 1, [2072].log_data[2].valid := 1, [2072].log_data[3].valid := 1, [2072].log_data[4].valid := 1, [2072].time.Year := 2022, [2072].time.Month := 5, [2072].time.Day := 1, [2072].time.Hour := 2, [2072].time.Minute := 14, [2072].time.Second := 59, [2072].time.DST_ON := 1, [2073].log_data[0].min := 1.0, [2073].log_data[0].max := 1.0, [2073].log_data[0].total := 300.0, [2073].log_data[0].time := 300.0, [2073].log_data[0].minminute := 15, [2073].log_data[0].maxminute := 15, [2073].log_data[0].valid := 1, [2073].log_data[1].valid := 1, [2073].log_data[2].valid := 1, [2073].log_data[3].valid := 1, [2073].log_data[4].valid := 1, [2073].time.Year := 2022, [2073].time.Month := 5, [2073].time.Day := 1, [2073].time.Hour := 2, [2073].time.Minute := 19, [2073].time.Second := 59, [2073].time.DST_ON := 1, [2074].log_data[0].min := 1.0, [2074].log_data[0].max := 1.0, [2074].log_data[0].total := 300.0, [2074].log_data[0].time := 300.0, [2074].log_data[0].minminute := 20,
        [2074].log_data[0].maxminute := 20, [2074].log_data[0].valid := 1, [2074].log_data[1].valid := 1, [2074].log_data[2].valid := 1, [2074].log_data[3].valid := 1, [2074].log_data[4].valid := 1, [2074].time.Year := 2022, [2074].time.Month := 5, [2074].time.Day := 1, [2074].time.Hour := 2, [2074].time.Minute := 24, [2074].time.Second := 59, [2074].time.DST_ON := 1, [2075].log_data[0].min := 1.0, [2075].log_data[0].max := 1.0, [2075].log_data[0].total := 300.0, [2075].log_data[0].time := 300.0, [2075].log_data[0].minminute := 25, [2075].log_data[0].maxminute := 25, [2075].log_data[0].valid := 1, [2075].log_data[1].valid := 1, [2075].log_data[2].valid := 1, [2075].log_data[3].valid := 1, [2075].log_data[4].valid := 1, [2075].time.Year := 2022, [2075].time.Month := 5, [2075].time.Day := 1, [2075].time.Hour := 2, [2075].time.Minute := 29, [2075].time.Second := 59, [2075].time.DST_ON := 1, [2076].log_data[0].min := 1.0, [2076].log_data[0].max := 1.0, [2076].log_data[0].total := 300.0, [2076].log_data[0].time := 300.0, [2076].log_data[0].minminute := 30, [2076].log_data[0].maxminute := 30, [2076].log_data[0].valid := 1, [2076].log_data[1].valid := 1, [2076].log_data[2].valid := 1, [2076].log_data[3].valid := 1, [2076].log_data[4].valid := 1, [2076].time.Year := 2022, [2076].time.Month := 5, [2076].time.Day := 1, [2076].time.Hour := 2, [2076].time.Minute := 34, [2076].time.Second := 59, [2076].time.DST_ON := 1, [2077].log_data[0].min := 1.0, [2077].log_data[0].max := 1.0, [2077].log_data[0].total := 300.0, [2077].log_data[0].time := 300.0, [2077].log_data[0].minminute := 35, [2077].log_data[0].maxminute := 35, [2077].log_data[0].valid := 1, [2077].log_data[1].valid := 1, [2077].log_data[2].valid := 1, [2077].log_data[3].valid := 1, [2077].log_data[4].valid := 1,
        [2077].time.Year := 2022, [2077].time.Month := 5, [2077].time.Day := 1, [2077].time.Hour := 2, [2077].time.Minute := 39, [2077].time.Second := 59, [2077].time.DST_ON := 1, [2078].log_data[0].min := 1.0, [2078].log_data[0].max := 1.0, [2078].log_data[0].total := 300.0, [2078].log_data[0].time := 300.0, [2078].log_data[0].minminute := 40, [2078].log_data[0].maxminute := 40, [2078].log_data[0].valid := 1, [2078].log_data[1].valid := 1, [2078].log_data[2].valid := 1, [2078].log_data[3].valid := 1, [2078].log_data[4].valid := 1, [2078].time.Year := 2022, [2078].time.Month := 5, [2078].time.Day := 1, [2078].time.Hour := 2, [2078].time.Minute := 44, [2078].time.Second := 59, [2078].time.DST_ON := 1, [2079].log_data[0].min := 1.0, [2079].log_data[0].max := 1.0, [2079].log_data[0].total := 300.0, [2079].log_data[0].time := 300.0, [2079].log_data[0].minminute := 45, [2079].log_data[0].maxminute := 45, [2079].log_data[0].valid := 1, [2079].log_data[1].valid := 1, [2079].log_data[2].valid := 1, [2079].log_data[3].valid := 1, [2079].log_data[4].valid := 1, [2079].time.Year := 2022, [2079].time.Month := 5, [2079].time.Day := 1, [2079].time.Hour := 2, [2079].time.Minute := 49, [2079].time.Second := 59, [2079].time.DST_ON := 1, [2080].log_data[0].min := 1.0, [2080].log_data[0].max := 1.0, [2080].log_data[0].total := 300.0, [2080].log_data[0].time := 300.0, [2080].log_data[0].minminute := 50, [2080].log_data[0].maxminute := 50, [2080].log_data[0].valid := 1, [2080].log_data[1].valid := 1, [2080].log_data[2].valid := 1, [2080].log_data[3].valid := 1, [2080].log_data[4].valid := 1, [2080].time.Year := 2022, [2080].time.Month := 5, [2080].time.Day := 1, [2080].time.Hour := 2, [2080].time.Minute := 54, [2080].time.Second := 59,
        [2080].time.DST_ON := 1, [2081].log_data[0].min := 1.0, [2081].log_data[0].max := 1.0, [2081].log_data[0].total := 300.0, [2081].log_data[0].time := 300.0, [2081].log_data[0].minminute := 55, [2081].log_data[0].maxminute := 55, [2081].log_data[0].valid := 1, [2081].log_data[1].valid := 1, [2081].log_data[2].valid := 1, [2081].log_data[3].valid := 1, [2081].log_data[4].valid := 1, [2081].time.Year := 2022, [2081].time.Month := 5, [2081].time.Day := 1, [2081].time.Hour := 2, [2081].time.Minute := 59, [2081].time.Second := 59, [2081].time.DST_ON := 1, [2082].log_data[0].min := 1.0, [2082].log_data[0].max := 1.0, [2082].log_data[0].total := 300.0, [2082].log_data[0].time := 300.0, [2082].log_data[0].valid := 1, [2082].log_data[1].valid := 1, [2082].log_data[2].valid := 1, [2082].log_data[3].valid := 1, [2082].log_data[4].valid := 1, [2082].time.Year := 2022, [2082].time.Month := 5, [2082].time.Day := 1, [2082].time.Hour := 3, [2082].time.Minute := 4, [2082].time.Second := 59, [2082].time.DST_ON := 1, [2083].log_data[0].min := 1.0, [2083].log_data[0].max := 1.0, [2083].log_data[0].total := 300.0, [2083].log_data[0].time := 300.0, [2083].log_data[0].minminute := 5, [2083].log_data[0].maxminute := 5, [2083].log_data[0].valid := 1, [2083].log_data[1].valid := 1, [2083].log_data[2].valid := 1, [2083].log_data[3].valid := 1, [2083].log_data[4].valid := 1, [2083].time.Year := 2022, [2083].time.Month := 5, [2083].time.Day := 1, [2083].time.Hour := 3, [2083].time.Minute := 9, [2083].time.Second := 59, [2083].time.DST_ON := 1, [2084].log_data[0].min := 1.0, [2084].log_data[0].max := 1.0, [2084].log_data[0].total := 300.0, [2084].log_data[0].time := 300.0, [2084].log_data[0].minminute := 10, [2084].log_data[0].maxminute := 10, [2084].log_data[0].valid := 1,
        [2084].log_data[1].valid := 1, [2084].log_data[2].valid := 1, [2084].log_data[3].valid := 1, [2084].log_data[4].valid := 1, [2084].time.Year := 2022, [2084].time.Month := 5, [2084].time.Day := 1, [2084].time.Hour := 3, [2084].time.Minute := 14, [2084].time.Second := 59, [2084].time.DST_ON := 1, [2085].log_data[0].min := 1.0, [2085].log_data[0].max := 1.0, [2085].log_data[0].total := 300.0, [2085].log_data[0].time := 300.0, [2085].log_data[0].minminute := 15, [2085].log_data[0].maxminute := 15, [2085].log_data[0].valid := 1, [2085].log_data[1].valid := 1, [2085].log_data[2].valid := 1, [2085].log_data[3].valid := 1, [2085].log_data[4].valid := 1, [2085].time.Year := 2022, [2085].time.Month := 5, [2085].time.Day := 1, [2085].time.Hour := 3, [2085].time.Minute := 19, [2085].time.Second := 59, [2085].time.DST_ON := 1, [2086].log_data[0].min := 1.0, [2086].log_data[0].max := 1.0, [2086].log_data[0].total := 300.0, [2086].log_data[0].time := 300.0, [2086].log_data[0].minminute := 20, [2086].log_data[0].maxminute := 20, [2086].log_data[0].valid := 1, [2086].log_data[1].valid := 1, [2086].log_data[2].valid := 1, [2086].log_data[3].valid := 1, [2086].log_data[4].valid := 1, [2086].time.Year := 2022, [2086].time.Month := 5, [2086].time.Day := 1, [2086].time.Hour := 3, [2086].time.Minute := 24, [2086].time.Second := 59, [2086].time.DST_ON := 1, [2087].log_data[0].min := 1.0, [2087].log_data[0].max := 1.0, [2087].log_data[0].total := 300.0, [2087].log_data[0].time := 300.0, [2087].log_data[0].minminute := 25, [2087].log_data[0].maxminute := 25, [2087].log_data[0].valid := 1, [2087].log_data[1].valid := 1, [2087].log_data[2].valid := 1, [2087].log_data[3].valid := 1, [2087].log_data[4].valid := 1, [2087].time.Year := 2022, [2087].time.Month := 5,
        [2087].time.Day := 1, [2087].time.Hour := 3, [2087].time.Minute := 29, [2087].time.Second := 59, [2087].time.DST_ON := 1, [2088].log_data[0].min := 1.0, [2088].log_data[0].max := 1.0, [2088].log_data[0].total := 300.0, [2088].log_data[0].time := 300.0, [2088].log_data[0].minminute := 30, [2088].log_data[0].maxminute := 30, [2088].log_data[0].valid := 1, [2088].log_data[1].valid := 1, [2088].log_data[2].valid := 1, [2088].log_data[3].valid := 1, [2088].log_data[4].valid := 1, [2088].time.Year := 2022, [2088].time.Month := 5, [2088].time.Day := 1, [2088].time.Hour := 3, [2088].time.Minute := 34, [2088].time.Second := 59, [2088].time.DST_ON := 1, [2089].log_data[0].min := 1.0, [2089].log_data[0].max := 1.0, [2089].log_data[0].total := 300.0, [2089].log_data[0].time := 300.0, [2089].log_data[0].minminute := 35, [2089].log_data[0].maxminute := 35, [2089].log_data[0].valid := 1, [2089].log_data[1].valid := 1, [2089].log_data[2].valid := 1, [2089].log_data[3].valid := 1, [2089].log_data[4].valid := 1, [2089].time.Year := 2022, [2089].time.Month := 5, [2089].time.Day := 1, [2089].time.Hour := 3, [2089].time.Minute := 39, [2089].time.Second := 59, [2089].time.DST_ON := 1, [2090].log_data[0].min := 1.0, [2090].log_data[0].max := 1.0, [2090].log_data[0].total := 299.999, [2090].log_data[0].time := 299.999, [2090].log_data[0].minminute := 40, [2090].log_data[0].maxminute := 40, [2090].log_data[0].valid := 1, [2090].log_data[1].valid := 1, [2090].log_data[2].valid := 1, [2090].log_data[3].valid := 1, [2090].log_data[4].valid := 1, [2090].time.Year := 2022, [2090].time.Month := 5, [2090].time.Day := 1, [2090].time.Hour := 3, [2090].time.Minute := 44, [2090].time.Second := 59, [2090].time.DST_ON := 1, [2091].log_data[0].min := 1.0,
        [2091].log_data[0].max := 1.0, [2091].log_data[0].total := 300.0, [2091].log_data[0].time := 300.0, [2091].log_data[0].minminute := 45, [2091].log_data[0].maxminute := 45, [2091].log_data[0].valid := 1, [2091].log_data[1].valid := 1, [2091].log_data[2].valid := 1, [2091].log_data[3].valid := 1, [2091].log_data[4].valid := 1, [2091].time.Year := 2022, [2091].time.Month := 5, [2091].time.Day := 1, [2091].time.Hour := 3, [2091].time.Minute := 49, [2091].time.Second := 59, [2091].time.DST_ON := 1, [2092].log_data[0].min := 1.0, [2092].log_data[0].max := 1.0, [2092].log_data[0].total := 300.0, [2092].log_data[0].time := 300.0, [2092].log_data[0].minminute := 50, [2092].log_data[0].maxminute := 50, [2092].log_data[0].valid := 1, [2092].log_data[1].valid := 1, [2092].log_data[2].valid := 1, [2092].log_data[3].valid := 1, [2092].log_data[4].valid := 1, [2092].time.Year := 2022, [2092].time.Month := 5, [2092].time.Day := 1, [2092].time.Hour := 3, [2092].time.Minute := 54, [2092].time.Second := 59, [2092].time.DST_ON := 1, [2093].log_data[0].min := 1.0, [2093].log_data[0].max := 1.0, [2093].log_data[0].total := 300.0, [2093].log_data[0].time := 300.0, [2093].log_data[0].minminute := 55, [2093].log_data[0].maxminute := 55, [2093].log_data[0].valid := 1, [2093].log_data[1].valid := 1, [2093].log_data[2].valid := 1, [2093].log_data[3].valid := 1, [2093].log_data[4].valid := 1, [2093].time.Year := 2022, [2093].time.Month := 5, [2093].time.Day := 1, [2093].time.Hour := 3, [2093].time.Minute := 59, [2093].time.Second := 59, [2093].time.DST_ON := 1, [2094].log_data[0].min := 1.0, [2094].log_data[0].max := 1.0, [2094].log_data[0].total := 300.0, [2094].log_data[0].time := 300.0, [2094].log_data[0].valid := 1, [2094].log_data[1].valid := 1, [2094].log_data[2].valid := 1,
        [2094].log_data[3].valid := 1, [2094].log_data[4].valid := 1, [2094].time.Year := 2022, [2094].time.Month := 5, [2094].time.Day := 1, [2094].time.Hour := 4, [2094].time.Minute := 4, [2094].time.Second := 59, [2094].time.DST_ON := 1, [2095].log_data[0].min := 1.0, [2095].log_data[0].max := 1.0, [2095].log_data[0].total := 300.0, [2095].log_data[0].time := 300.0, [2095].log_data[0].minminute := 5, [2095].log_data[0].maxminute := 5, [2095].log_data[0].valid := 1, [2095].log_data[1].valid := 1, [2095].log_data[2].valid := 1, [2095].log_data[3].valid := 1, [2095].log_data[4].valid := 1, [2095].time.Year := 2022, [2095].time.Month := 5, [2095].time.Day := 1, [2095].time.Hour := 4, [2095].time.Minute := 9, [2095].time.Second := 59, [2095].time.DST_ON := 1, [2096].log_data[0].min := 1.0, [2096].log_data[0].max := 1.0, [2096].log_data[0].total := 300.0, [2096].log_data[0].time := 300.0, [2096].log_data[0].minminute := 10, [2096].log_data[0].maxminute := 10, [2096].log_data[0].valid := 1, [2096].log_data[1].valid := 1, [2096].log_data[2].valid := 1, [2096].log_data[3].valid := 1, [2096].log_data[4].valid := 1, [2096].time.Year := 2022, [2096].time.Month := 5, [2096].time.Day := 1, [2096].time.Hour := 4, [2096].time.Minute := 14, [2096].time.Second := 59, [2096].time.DST_ON := 1, [2097].log_data[0].min := 1.0, [2097].log_data[0].max := 1.0, [2097].log_data[0].total := 299.999, [2097].log_data[0].time := 299.999, [2097].log_data[0].minminute := 15, [2097].log_data[0].maxminute := 15, [2097].log_data[0].valid := 1, [2097].log_data[1].valid := 1, [2097].log_data[2].valid := 1, [2097].log_data[3].valid := 1, [2097].log_data[4].valid := 1, [2097].time.Year := 2022, [2097].time.Month := 5, [2097].time.Day := 1, [2097].time.Hour := 4,
        [2097].time.Minute := 19, [2097].time.Second := 59, [2097].time.DST_ON := 1, [2098].log_data[0].min := 1.0, [2098].log_data[0].max := 1.0, [2098].log_data[0].total := 300.0, [2098].log_data[0].time := 300.0, [2098].log_data[0].minminute := 20, [2098].log_data[0].maxminute := 20, [2098].log_data[0].valid := 1, [2098].log_data[1].valid := 1, [2098].log_data[2].valid := 1, [2098].log_data[3].valid := 1, [2098].log_data[4].valid := 1, [2098].time.Year := 2022, [2098].time.Month := 5, [2098].time.Day := 1, [2098].time.Hour := 4, [2098].time.Minute := 24, [2098].time.Second := 59, [2098].time.DST_ON := 1, [2099].log_data[0].min := 1.0, [2099].log_data[0].max := 1.0, [2099].log_data[0].total := 300.0, [2099].log_data[0].time := 300.0, [2099].log_data[0].minminute := 25, [2099].log_data[0].maxminute := 25, [2099].log_data[0].valid := 1, [2099].log_data[1].valid := 1, [2099].log_data[2].valid := 1, [2099].log_data[3].valid := 1, [2099].log_data[4].valid := 1, [2099].time.Year := 2022, [2099].time.Month := 5, [2099].time.Day := 1, [2099].time.Hour := 4, [2099].time.Minute := 29, [2099].time.Second := 59, [2099].time.DST_ON := 1, [2100].log_data[0].min := 1.0, [2100].log_data[0].max := 1.0, [2100].log_data[0].total := 300.0, [2100].log_data[0].time := 300.0, [2100].log_data[0].minminute := 30, [2100].log_data[0].maxminute := 30, [2100].log_data[0].valid := 1, [2100].log_data[1].valid := 1, [2100].log_data[2].valid := 1, [2100].log_data[3].valid := 1, [2100].log_data[4].valid := 1, [2100].time.Year := 2022, [2100].time.Month := 5, [2100].time.Day := 1, [2100].time.Hour := 4, [2100].time.Minute := 34, [2100].time.Second := 59, [2100].time.DST_ON := 1, [2101].log_data[0].min := 1.0, [2101].log_data[0].max := 1.0, [2101].log_data[0].total := 300.0,
        [2101].log_data[0].time := 300.0, [2101].log_data[0].minminute := 35, [2101].log_data[0].maxminute := 35, [2101].log_data[0].valid := 1, [2101].log_data[1].valid := 1, [2101].log_data[2].valid := 1, [2101].log_data[3].valid := 1, [2101].log_data[4].valid := 1, [2101].time.Year := 2022, [2101].time.Month := 5, [2101].time.Day := 1, [2101].time.Hour := 4, [2101].time.Minute := 39, [2101].time.Second := 59, [2101].time.DST_ON := 1, [2102].log_data[0].min := 1.0, [2102].log_data[0].max := 1.0, [2102].log_data[0].total := 300.0, [2102].log_data[0].time := 300.0, [2102].log_data[0].minminute := 40, [2102].log_data[0].maxminute := 40, [2102].log_data[0].valid := 1, [2102].log_data[1].valid := 1, [2102].log_data[2].valid := 1, [2102].log_data[3].valid := 1, [2102].log_data[4].valid := 1, [2102].time.Year := 2022, [2102].time.Month := 5, [2102].time.Day := 1, [2102].time.Hour := 4, [2102].time.Minute := 44, [2102].time.Second := 59, [2102].time.DST_ON := 1, [2103].log_data[0].min := 1.0, [2103].log_data[0].max := 1.0, [2103].log_data[0].total := 300.0, [2103].log_data[0].time := 300.0, [2103].log_data[0].minminute := 45, [2103].log_data[0].maxminute := 45, [2103].log_data[0].valid := 1, [2103].log_data[1].valid := 1, [2103].log_data[2].valid := 1, [2103].log_data[3].valid := 1, [2103].log_data[4].valid := 1, [2103].time.Year := 2022, [2103].time.Month := 5, [2103].time.Day := 1, [2103].time.Hour := 4, [2103].time.Minute := 49, [2103].time.Second := 59, [2103].time.DST_ON := 1, [2104].log_data[0].min := 1.0, [2104].log_data[0].max := 1.0, [2104].log_data[0].total := 300.0, [2104].log_data[0].time := 300.0, [2104].log_data[0].minminute := 50, [2104].log_data[0].maxminute := 50, [2104].log_data[0].valid := 1, [2104].log_data[1].valid := 1, [2104].log_data[2].valid := 1,
        [2104].log_data[3].valid := 1, [2104].log_data[4].valid := 1, [2104].time.Year := 2022, [2104].time.Month := 5, [2104].time.Day := 1, [2104].time.Hour := 4, [2104].time.Minute := 54, [2104].time.Second := 59, [2104].time.DST_ON := 1, [2105].log_data[0].min := 1.0, [2105].log_data[0].max := 1.0, [2105].log_data[0].total := 300.0, [2105].log_data[0].time := 300.0, [2105].log_data[0].minminute := 55, [2105].log_data[0].maxminute := 55, [2105].log_data[0].valid := 1, [2105].log_data[1].valid := 1, [2105].log_data[2].valid := 1, [2105].log_data[3].valid := 1, [2105].log_data[4].valid := 1, [2105].time.Year := 2022, [2105].time.Month := 5, [2105].time.Day := 1, [2105].time.Hour := 4, [2105].time.Minute := 59, [2105].time.Second := 59, [2105].time.DST_ON := 1, [2106].log_data[0].min := 1.0, [2106].log_data[0].max := 1.0, [2106].log_data[0].total := 300.0, [2106].log_data[0].time := 300.0, [2106].log_data[0].valid := 1, [2106].log_data[1].valid := 1, [2106].log_data[2].valid := 1, [2106].log_data[3].valid := 1, [2106].log_data[4].valid := 1, [2106].time.Year := 2022, [2106].time.Month := 5, [2106].time.Day := 1, [2106].time.Hour := 5, [2106].time.Minute := 4, [2106].time.Second := 59, [2106].time.DST_ON := 1, [2107].log_data[0].min := 1.0, [2107].log_data[0].max := 1.0, [2107].log_data[0].total := 300.0, [2107].log_data[0].time := 300.0, [2107].log_data[0].minminute := 5, [2107].log_data[0].maxminute := 5, [2107].log_data[0].valid := 1, [2107].log_data[1].valid := 1, [2107].log_data[2].valid := 1, [2107].log_data[3].valid := 1, [2107].log_data[4].valid := 1, [2107].time.Year := 2022, [2107].time.Month := 5, [2107].time.Day := 1, [2107].time.Hour := 5, [2107].time.Minute := 9, [2107].time.Second := 59,
        [2107].time.DST_ON := 1, [2108].log_data[0].min := 1.0, [2108].log_data[0].max := 1.0, [2108].log_data[0].total := 300.0, [2108].log_data[0].time := 300.0, [2108].log_data[0].minminute := 10, [2108].log_data[0].maxminute := 10, [2108].log_data[0].valid := 1, [2108].log_data[1].valid := 1, [2108].log_data[2].valid := 1, [2108].log_data[3].valid := 1, [2108].log_data[4].valid := 1, [2108].time.Year := 2022, [2108].time.Month := 5, [2108].time.Day := 1, [2108].time.Hour := 5, [2108].time.Minute := 14, [2108].time.Second := 59, [2108].time.DST_ON := 1, [2109].log_data[0].min := 1.0, [2109].log_data[0].max := 1.0, [2109].log_data[0].total := 300.0, [2109].log_data[0].time := 300.0, [2109].log_data[0].minminute := 15, [2109].log_data[0].maxminute := 15, [2109].log_data[0].valid := 1, [2109].log_data[1].valid := 1, [2109].log_data[2].valid := 1, [2109].log_data[3].valid := 1, [2109].log_data[4].valid := 1, [2109].time.Year := 2022, [2109].time.Month := 5, [2109].time.Day := 1, [2109].time.Hour := 5, [2109].time.Minute := 19, [2109].time.Second := 59, [2109].time.DST_ON := 1, [2110].log_data[0].min := 1.0, [2110].log_data[0].max := 1.0, [2110].log_data[0].total := 300.0, [2110].log_data[0].time := 300.0, [2110].log_data[0].minminute := 20, [2110].log_data[0].maxminute := 20, [2110].log_data[0].valid := 1, [2110].log_data[1].valid := 1, [2110].log_data[2].valid := 1, [2110].log_data[3].valid := 1, [2110].log_data[4].valid := 1, [2110].time.Year := 2022, [2110].time.Month := 5, [2110].time.Day := 1, [2110].time.Hour := 5, [2110].time.Minute := 24, [2110].time.Second := 59, [2110].time.DST_ON := 1, [2111].log_data[0].min := 1.0, [2111].log_data[0].max := 1.0, [2111].log_data[0].total := 300.0, [2111].log_data[0].time := 300.0, [2111].log_data[0].minminute := 25,
        [2111].log_data[0].maxminute := 25, [2111].log_data[0].valid := 1, [2111].log_data[1].valid := 1, [2111].log_data[2].valid := 1, [2111].log_data[3].valid := 1, [2111].log_data[4].valid := 1, [2111].time.Year := 2022, [2111].time.Month := 5, [2111].time.Day := 1, [2111].time.Hour := 5, [2111].time.Minute := 29, [2111].time.Second := 59, [2111].time.DST_ON := 1, [2112].log_data[0].min := 1.0, [2112].log_data[0].max := 1.0, [2112].log_data[0].total := 300.0, [2112].log_data[0].time := 300.0, [2112].log_data[0].minminute := 30, [2112].log_data[0].maxminute := 30, [2112].log_data[0].valid := 1, [2112].log_data[1].valid := 1, [2112].log_data[2].valid := 1, [2112].log_data[3].valid := 1, [2112].log_data[4].valid := 1, [2112].time.Year := 2022, [2112].time.Month := 5, [2112].time.Day := 1, [2112].time.Hour := 5, [2112].time.Minute := 34, [2112].time.Second := 59, [2112].time.DST_ON := 1, [2113].log_data[0].min := 1.0, [2113].log_data[0].max := 1.0, [2113].log_data[0].total := 300.0, [2113].log_data[0].time := 300.0, [2113].log_data[0].minminute := 35, [2113].log_data[0].maxminute := 35, [2113].log_data[0].valid := 1, [2113].log_data[1].valid := 1, [2113].log_data[2].valid := 1, [2113].log_data[3].valid := 1, [2113].log_data[4].valid := 1, [2113].time.Year := 2022, [2113].time.Month := 5, [2113].time.Day := 1, [2113].time.Hour := 5, [2113].time.Minute := 39, [2113].time.Second := 59, [2113].time.DST_ON := 1, [2114].log_data[0].min := 1.0, [2114].log_data[0].max := 1.0, [2114].log_data[0].total := 300.0, [2114].log_data[0].time := 300.0, [2114].log_data[0].minminute := 40, [2114].log_data[0].maxminute := 40, [2114].log_data[0].valid := 1, [2114].log_data[1].valid := 1, [2114].log_data[2].valid := 1, [2114].log_data[3].valid := 1, [2114].log_data[4].valid := 1,
        [2114].time.Year := 2022, [2114].time.Month := 5, [2114].time.Day := 1, [2114].time.Hour := 5, [2114].time.Minute := 44, [2114].time.Second := 59, [2114].time.DST_ON := 1, [2115].log_data[0].min := 1.0, [2115].log_data[0].max := 1.0, [2115].log_data[0].total := 299.999, [2115].log_data[0].time := 299.999, [2115].log_data[0].minminute := 45, [2115].log_data[0].maxminute := 45, [2115].log_data[0].valid := 1, [2115].log_data[1].valid := 1, [2115].log_data[2].valid := 1, [2115].log_data[3].valid := 1, [2115].log_data[4].valid := 1, [2115].time.Year := 2022, [2115].time.Month := 5, [2115].time.Day := 1, [2115].time.Hour := 5, [2115].time.Minute := 49, [2115].time.Second := 59, [2115].time.DST_ON := 1, [2116].log_data[0].min := 1.0, [2116].log_data[0].max := 1.0, [2116].log_data[0].total := 300.0, [2116].log_data[0].time := 300.0, [2116].log_data[0].minminute := 50, [2116].log_data[0].maxminute := 50, [2116].log_data[0].valid := 1, [2116].log_data[1].valid := 1, [2116].log_data[2].valid := 1, [2116].log_data[3].valid := 1, [2116].log_data[4].valid := 1, [2116].time.Year := 2022, [2116].time.Month := 5, [2116].time.Day := 1, [2116].time.Hour := 5, [2116].time.Minute := 54, [2116].time.Second := 59, [2116].time.DST_ON := 1, [2117].log_data[0].min := 1.0, [2117].log_data[0].max := 1.0, [2117].log_data[0].total := 300.0, [2117].log_data[0].time := 300.0, [2117].log_data[0].minminute := 55, [2117].log_data[0].maxminute := 55, [2117].log_data[0].valid := 1, [2117].log_data[1].valid := 1, [2117].log_data[2].valid := 1, [2117].log_data[3].valid := 1, [2117].log_data[4].valid := 1, [2117].time.Year := 2022, [2117].time.Month := 5, [2117].time.Day := 1, [2117].time.Hour := 5, [2117].time.Minute := 59, [2117].time.Second := 59,
        [2117].time.DST_ON := 1, [2118].log_data[0].min := 1.0, [2118].log_data[0].max := 1.0, [2118].log_data[0].total := 300.0, [2118].log_data[0].time := 300.0, [2118].log_data[0].valid := 1, [2118].log_data[1].valid := 1, [2118].log_data[2].valid := 1, [2118].log_data[3].valid := 1, [2118].log_data[4].valid := 1, [2118].time.Year := 2022, [2118].time.Month := 5, [2118].time.Day := 1, [2118].time.Hour := 6, [2118].time.Minute := 4, [2118].time.Second := 59, [2118].time.DST_ON := 1, [2119].log_data[0].min := 1.0, [2119].log_data[0].max := 1.0, [2119].log_data[0].total := 300.0, [2119].log_data[0].time := 300.0, [2119].log_data[0].minminute := 5, [2119].log_data[0].maxminute := 5, [2119].log_data[0].valid := 1, [2119].log_data[1].valid := 1, [2119].log_data[2].valid := 1, [2119].log_data[3].valid := 1, [2119].log_data[4].valid := 1, [2119].time.Year := 2022, [2119].time.Month := 5, [2119].time.Day := 1, [2119].time.Hour := 6, [2119].time.Minute := 9, [2119].time.Second := 59, [2119].time.DST_ON := 1, [2120].log_data[0].min := 1.0, [2120].log_data[0].max := 1.0, [2120].log_data[0].total := 300.0, [2120].log_data[0].time := 300.0, [2120].log_data[0].minminute := 10, [2120].log_data[0].maxminute := 10, [2120].log_data[0].valid := 1, [2120].log_data[1].valid := 1, [2120].log_data[2].valid := 1, [2120].log_data[3].valid := 1, [2120].log_data[4].valid := 1, [2120].time.Year := 2022, [2120].time.Month := 5, [2120].time.Day := 1, [2120].time.Hour := 6, [2120].time.Minute := 14, [2120].time.Second := 59, [2120].time.DST_ON := 1, [2121].log_data[0].min := 1.0, [2121].log_data[0].max := 1.0, [2121].log_data[0].total := 300.0, [2121].log_data[0].time := 300.0, [2121].log_data[0].minminute := 15, [2121].log_data[0].maxminute := 15, [2121].log_data[0].valid := 1,
        [2121].log_data[1].valid := 1, [2121].log_data[2].valid := 1, [2121].log_data[3].valid := 1, [2121].log_data[4].valid := 1, [2121].time.Year := 2022, [2121].time.Month := 5, [2121].time.Day := 1, [2121].time.Hour := 6, [2121].time.Minute := 19, [2121].time.Second := 59, [2121].time.DST_ON := 1, [2122].log_data[0].min := 1.0, [2122].log_data[0].max := 1.0, [2122].log_data[0].total := 300.0, [2122].log_data[0].time := 300.0, [2122].log_data[0].minminute := 20, [2122].log_data[0].maxminute := 20, [2122].log_data[0].valid := 1, [2122].log_data[1].valid := 1, [2122].log_data[2].valid := 1, [2122].log_data[3].valid := 1, [2122].log_data[4].valid := 1, [2122].time.Year := 2022, [2122].time.Month := 5, [2122].time.Day := 1, [2122].time.Hour := 6, [2122].time.Minute := 24, [2122].time.Second := 59, [2122].time.DST_ON := 1, [2123].log_data[0].min := 1.0, [2123].log_data[0].max := 1.0, [2123].log_data[0].total := 300.0, [2123].log_data[0].time := 300.0, [2123].log_data[0].minminute := 25, [2123].log_data[0].maxminute := 25, [2123].log_data[0].valid := 1, [2123].log_data[1].valid := 1, [2123].log_data[2].valid := 1, [2123].log_data[3].valid := 1, [2123].log_data[4].valid := 1, [2123].time.Year := 2022, [2123].time.Month := 5, [2123].time.Day := 1, [2123].time.Hour := 6, [2123].time.Minute := 29, [2123].time.Second := 59, [2123].time.DST_ON := 1, [2124].log_data[0].min := 1.0, [2124].log_data[0].max := 1.0, [2124].log_data[0].total := 300.0, [2124].log_data[0].time := 300.0, [2124].log_data[0].minminute := 30, [2124].log_data[0].maxminute := 30, [2124].log_data[0].valid := 1, [2124].log_data[1].valid := 1, [2124].log_data[2].valid := 1, [2124].log_data[3].valid := 1, [2124].log_data[4].valid := 1, [2124].time.Year := 2022, [2124].time.Month := 5,
        [2124].time.Day := 1, [2124].time.Hour := 6, [2124].time.Minute := 34, [2124].time.Second := 59, [2124].time.DST_ON := 1, [2125].log_data[0].min := 1.0, [2125].log_data[0].max := 1.0, [2125].log_data[0].total := 300.0, [2125].log_data[0].time := 300.0, [2125].log_data[0].minminute := 35, [2125].log_data[0].maxminute := 35, [2125].log_data[0].valid := 1, [2125].log_data[1].valid := 1, [2125].log_data[2].valid := 1, [2125].log_data[3].valid := 1, [2125].log_data[4].valid := 1, [2125].time.Year := 2022, [2125].time.Month := 5, [2125].time.Day := 1, [2125].time.Hour := 6, [2125].time.Minute := 39, [2125].time.Second := 59, [2125].time.DST_ON := 1, [2126].log_data[0].min := 1.0, [2126].log_data[0].max := 1.0, [2126].log_data[0].total := 300.0, [2126].log_data[0].time := 300.0, [2126].log_data[0].minminute := 40, [2126].log_data[0].maxminute := 40, [2126].log_data[0].valid := 1, [2126].log_data[1].valid := 1, [2126].log_data[2].valid := 1, [2126].log_data[3].valid := 1, [2126].log_data[4].valid := 1, [2126].time.Year := 2022, [2126].time.Month := 5, [2126].time.Day := 1, [2126].time.Hour := 6, [2126].time.Minute := 44, [2126].time.Second := 59, [2126].time.DST_ON := 1, [2127].log_data[0].min := 1.0, [2127].log_data[0].max := 1.0, [2127].log_data[0].total := 300.0, [2127].log_data[0].time := 300.0, [2127].log_data[0].minminute := 45, [2127].log_data[0].maxminute := 45, [2127].log_data[0].valid := 1, [2127].log_data[1].valid := 1, [2127].log_data[2].valid := 1, [2127].log_data[3].valid := 1, [2127].log_data[4].valid := 1, [2127].time.Year := 2022, [2127].time.Month := 5, [2127].time.Day := 1, [2127].time.Hour := 6, [2127].time.Minute := 49, [2127].time.Second := 59, [2127].time.DST_ON := 1, [2128].log_data[0].min := 1.0,
        [2128].log_data[0].max := 1.0, [2128].log_data[0].total := 300.0, [2128].log_data[0].time := 300.0, [2128].log_data[0].minminute := 50, [2128].log_data[0].maxminute := 50, [2128].log_data[0].valid := 1, [2128].log_data[1].valid := 1, [2128].log_data[2].valid := 1, [2128].log_data[3].valid := 1, [2128].log_data[4].valid := 1, [2128].time.Year := 2022, [2128].time.Month := 5, [2128].time.Day := 1, [2128].time.Hour := 6, [2128].time.Minute := 54, [2128].time.Second := 59, [2128].time.DST_ON := 1, [2129].log_data[0].min := 1.0, [2129].log_data[0].max := 1.0, [2129].log_data[0].total := 300.0, [2129].log_data[0].time := 300.0, [2129].log_data[0].minminute := 55, [2129].log_data[0].maxminute := 55, [2129].log_data[0].valid := 1, [2129].log_data[1].valid := 1, [2129].log_data[2].valid := 1, [2129].log_data[3].valid := 1, [2129].log_data[4].valid := 1, [2129].time.Year := 2022, [2129].time.Month := 5, [2129].time.Day := 1, [2129].time.Hour := 6, [2129].time.Minute := 59, [2129].time.Second := 59, [2129].time.DST_ON := 1, [2130].log_data[0].min := 1.0, [2130].log_data[0].max := 1.0, [2130].log_data[0].total := 300.0, [2130].log_data[0].time := 300.0, [2130].log_data[0].valid := 1, [2130].log_data[1].valid := 1, [2130].log_data[2].valid := 1, [2130].log_data[3].valid := 1, [2130].log_data[4].valid := 1, [2130].time.Year := 2022, [2130].time.Month := 5, [2130].time.Day := 1, [2130].time.Hour := 7, [2130].time.Minute := 4, [2130].time.Second := 59, [2130].time.DST_ON := 1, [2131].log_data[0].min := 1.0, [2131].log_data[0].max := 1.0, [2131].log_data[0].total := 300.0, [2131].log_data[0].time := 300.0, [2131].log_data[0].minminute := 5, [2131].log_data[0].maxminute := 5, [2131].log_data[0].valid := 1, [2131].log_data[1].valid := 1, [2131].log_data[2].valid := 1,
        [2131].log_data[3].valid := 1, [2131].log_data[4].valid := 1, [2131].time.Year := 2022, [2131].time.Month := 5, [2131].time.Day := 1, [2131].time.Hour := 7, [2131].time.Minute := 9, [2131].time.Second := 59, [2131].time.DST_ON := 1, [2132].log_data[0].min := 1.0, [2132].log_data[0].max := 1.0, [2132].log_data[0].total := 300.0, [2132].log_data[0].time := 300.0, [2132].log_data[0].minminute := 10, [2132].log_data[0].maxminute := 10, [2132].log_data[0].valid := 1, [2132].log_data[1].valid := 1, [2132].log_data[2].valid := 1, [2132].log_data[3].valid := 1, [2132].log_data[4].valid := 1, [2132].time.Year := 2022, [2132].time.Month := 5, [2132].time.Day := 1, [2132].time.Hour := 7, [2132].time.Minute := 14, [2132].time.Second := 59, [2132].time.DST_ON := 1, [2133].log_data[0].min := 1.0, [2133].log_data[0].max := 1.0, [2133].log_data[0].total := 300.0, [2133].log_data[0].time := 300.0, [2133].log_data[0].minminute := 15, [2133].log_data[0].maxminute := 15, [2133].log_data[0].valid := 1, [2133].log_data[1].valid := 1, [2133].log_data[2].valid := 1, [2133].log_data[3].valid := 1, [2133].log_data[4].valid := 1, [2133].time.Year := 2022, [2133].time.Month := 5, [2133].time.Day := 1, [2133].time.Hour := 7, [2133].time.Minute := 19, [2133].time.Second := 59, [2133].time.DST_ON := 1, [2134].log_data[0].min := 1.0, [2134].log_data[0].max := 1.0, [2134].log_data[0].total := 300.0, [2134].log_data[0].time := 300.0, [2134].log_data[0].minminute := 20, [2134].log_data[0].maxminute := 20, [2134].log_data[0].valid := 1, [2134].log_data[1].valid := 1, [2134].log_data[2].valid := 1, [2134].log_data[3].valid := 1, [2134].log_data[4].valid := 1, [2134].time.Year := 2022, [2134].time.Month := 5, [2134].time.Day := 1, [2134].time.Hour := 7,
        [2134].time.Minute := 24, [2134].time.Second := 59, [2134].time.DST_ON := 1, [2135].log_data[0].min := 1.0, [2135].log_data[0].max := 1.0, [2135].log_data[0].total := 300.0, [2135].log_data[0].time := 300.0, [2135].log_data[0].minminute := 25, [2135].log_data[0].maxminute := 25, [2135].log_data[0].valid := 1, [2135].log_data[1].valid := 1, [2135].log_data[2].valid := 1, [2135].log_data[3].valid := 1, [2135].log_data[4].valid := 1, [2135].time.Year := 2022, [2135].time.Month := 5, [2135].time.Day := 1, [2135].time.Hour := 7, [2135].time.Minute := 29, [2135].time.Second := 59, [2135].time.DST_ON := 1, [2136].log_data[0].min := 1.0, [2136].log_data[0].max := 1.0, [2136].log_data[0].total := 300.0, [2136].log_data[0].time := 300.0, [2136].log_data[0].minminute := 30, [2136].log_data[0].maxminute := 30, [2136].log_data[0].valid := 1, [2136].log_data[1].valid := 1, [2136].log_data[2].valid := 1, [2136].log_data[3].valid := 1, [2136].log_data[4].valid := 1, [2136].time.Year := 2022, [2136].time.Month := 5, [2136].time.Day := 1, [2136].time.Hour := 7, [2136].time.Minute := 34, [2136].time.Second := 59, [2136].time.DST_ON := 1, [2137].log_data[0].min := 1.0, [2137].log_data[0].max := 1.0, [2137].log_data[0].total := 300.0, [2137].log_data[0].time := 300.0, [2137].log_data[0].minminute := 35, [2137].log_data[0].maxminute := 35, [2137].log_data[0].valid := 1, [2137].log_data[1].valid := 1, [2137].log_data[2].valid := 1, [2137].log_data[3].valid := 1, [2137].log_data[4].valid := 1, [2137].time.Year := 2022, [2137].time.Month := 5, [2137].time.Day := 1, [2137].time.Hour := 7, [2137].time.Minute := 39, [2137].time.Second := 59, [2137].time.DST_ON := 1, [2138].log_data[0].min := 1.0, [2138].log_data[0].max := 1.0, [2138].log_data[0].total := 300.0,
        [2138].log_data[0].time := 300.0, [2138].log_data[0].minminute := 40, [2138].log_data[0].maxminute := 40, [2138].log_data[0].valid := 1, [2138].log_data[1].valid := 1, [2138].log_data[2].valid := 1, [2138].log_data[3].valid := 1, [2138].log_data[4].valid := 1, [2138].time.Year := 2022, [2138].time.Month := 5, [2138].time.Day := 1, [2138].time.Hour := 7, [2138].time.Minute := 44, [2138].time.Second := 59, [2138].time.DST_ON := 1, [2139].log_data[0].min := 1.0, [2139].log_data[0].max := 1.0, [2139].log_data[0].total := 300.0, [2139].log_data[0].time := 300.0, [2139].log_data[0].minminute := 45, [2139].log_data[0].maxminute := 45, [2139].log_data[0].valid := 1, [2139].log_data[1].valid := 1, [2139].log_data[2].valid := 1, [2139].log_data[3].valid := 1, [2139].log_data[4].valid := 1, [2139].time.Year := 2022, [2139].time.Month := 5, [2139].time.Day := 1, [2139].time.Hour := 7, [2139].time.Minute := 49, [2139].time.Second := 59, [2139].time.DST_ON := 1, [2140].log_data[0].min := 1.0, [2140].log_data[0].max := 1.0, [2140].log_data[0].total := 300.0, [2140].log_data[0].time := 300.0, [2140].log_data[0].minminute := 50, [2140].log_data[0].maxminute := 50, [2140].log_data[0].valid := 1, [2140].log_data[1].valid := 1, [2140].log_data[2].valid := 1, [2140].log_data[3].valid := 1, [2140].log_data[4].valid := 1, [2140].time.Year := 2022, [2140].time.Month := 5, [2140].time.Day := 1, [2140].time.Hour := 7, [2140].time.Minute := 54, [2140].time.Second := 59, [2140].time.DST_ON := 1, [2141].log_data[0].min := 1.0, [2141].log_data[0].max := 1.0, [2141].log_data[0].total := 300.0, [2141].log_data[0].time := 300.0, [2141].log_data[0].minminute := 55, [2141].log_data[0].maxminute := 55, [2141].log_data[0].valid := 1, [2141].log_data[1].valid := 1, [2141].log_data[2].valid := 1,
        [2141].log_data[3].valid := 1, [2141].log_data[4].valid := 1, [2141].time.Year := 2022, [2141].time.Month := 5, [2141].time.Day := 1, [2141].time.Hour := 7, [2141].time.Minute := 59, [2141].time.Second := 59, [2141].time.DST_ON := 1, [2142].log_data[0].min := 1.0, [2142].log_data[0].max := 1.0, [2142].log_data[0].total := 300.0, [2142].log_data[0].time := 300.0, [2142].log_data[0].valid := 1, [2142].log_data[1].valid := 1, [2142].log_data[2].valid := 1, [2142].log_data[3].valid := 1, [2142].log_data[4].valid := 1, [2142].time.Year := 2022, [2142].time.Month := 5, [2142].time.Day := 1, [2142].time.Hour := 8, [2142].time.Minute := 4, [2142].time.Second := 59, [2142].time.DST_ON := 1, [2143].log_data[0].min := 1.0, [2143].log_data[0].max := 1.0, [2143].log_data[0].total := 300.0, [2143].log_data[0].time := 300.0, [2143].log_data[0].minminute := 5, [2143].log_data[0].maxminute := 5, [2143].log_data[0].valid := 1, [2143].log_data[1].valid := 1, [2143].log_data[2].valid := 1, [2143].log_data[3].valid := 1, [2143].log_data[4].valid := 1, [2143].time.Year := 2022, [2143].time.Month := 5, [2143].time.Day := 1, [2143].time.Hour := 8, [2143].time.Minute := 9, [2143].time.Second := 59, [2143].time.DST_ON := 1, [2144].log_data[0].min := 1.0, [2144].log_data[0].max := 1.0, [2144].log_data[0].total := 300.0, [2144].log_data[0].time := 300.0, [2144].log_data[0].minminute := 10, [2144].log_data[0].maxminute := 10, [2144].log_data[0].valid := 1, [2144].log_data[1].valid := 1, [2144].log_data[2].valid := 1, [2144].log_data[3].valid := 1, [2144].log_data[4].valid := 1, [2144].time.Year := 2022, [2144].time.Month := 5, [2144].time.Day := 1, [2144].time.Hour := 8, [2144].time.Minute := 14, [2144].time.Second := 59,
        [2144].time.DST_ON := 1, [2145].log_data[0].min := 1.0, [2145].log_data[0].max := 1.0, [2145].log_data[0].total := 300.0, [2145].log_data[0].time := 300.0, [2145].log_data[0].minminute := 15, [2145].log_data[0].maxminute := 15, [2145].log_data[0].valid := 1, [2145].log_data[1].valid := 1, [2145].log_data[2].valid := 1, [2145].log_data[3].valid := 1, [2145].log_data[4].valid := 1, [2145].time.Year := 2022, [2145].time.Month := 5, [2145].time.Day := 1, [2145].time.Hour := 8, [2145].time.Minute := 19, [2145].time.Second := 59, [2145].time.DST_ON := 1, [2146].log_data[0].min := 1.0, [2146].log_data[0].max := 1.0, [2146].log_data[0].total := 300.0, [2146].log_data[0].time := 300.0, [2146].log_data[0].minminute := 20, [2146].log_data[0].maxminute := 20, [2146].log_data[0].valid := 1, [2146].log_data[1].valid := 1, [2146].log_data[2].valid := 1, [2146].log_data[3].valid := 1, [2146].log_data[4].valid := 1, [2146].time.Year := 2022, [2146].time.Month := 5, [2146].time.Day := 1, [2146].time.Hour := 8, [2146].time.Minute := 24, [2146].time.Second := 59, [2146].time.DST_ON := 1, [2147].log_data[0].min := 1.0, [2147].log_data[0].max := 1.0, [2147].log_data[0].total := 300.0, [2147].log_data[0].time := 300.0, [2147].log_data[0].minminute := 25, [2147].log_data[0].maxminute := 25, [2147].log_data[0].valid := 1, [2147].log_data[1].valid := 1, [2147].log_data[2].valid := 1, [2147].log_data[3].valid := 1, [2147].log_data[4].valid := 1, [2147].time.Year := 2022, [2147].time.Month := 5, [2147].time.Day := 1, [2147].time.Hour := 8, [2147].time.Minute := 29, [2147].time.Second := 59, [2147].time.DST_ON := 1, [2148].log_data[0].min := 1.0, [2148].log_data[0].max := 1.0, [2148].log_data[0].total := 300.0, [2148].log_data[0].time := 300.0, [2148].log_data[0].minminute := 30,
        [2148].log_data[0].maxminute := 30, [2148].log_data[0].valid := 1, [2148].log_data[1].valid := 1, [2148].log_data[2].valid := 1, [2148].log_data[3].valid := 1, [2148].log_data[4].valid := 1, [2148].time.Year := 2022, [2148].time.Month := 5, [2148].time.Day := 1, [2148].time.Hour := 8, [2148].time.Minute := 34, [2148].time.Second := 59, [2148].time.DST_ON := 1, [2149].log_data[0].min := 1.0, [2149].log_data[0].max := 1.0, [2149].log_data[0].total := 300.0, [2149].log_data[0].time := 300.0, [2149].log_data[0].minminute := 35, [2149].log_data[0].maxminute := 35, [2149].log_data[0].valid := 1, [2149].log_data[1].valid := 1, [2149].log_data[2].valid := 1, [2149].log_data[3].valid := 1, [2149].log_data[4].valid := 1, [2149].time.Year := 2022, [2149].time.Month := 5, [2149].time.Day := 1, [2149].time.Hour := 8, [2149].time.Minute := 39, [2149].time.Second := 59, [2149].time.DST_ON := 1, [2150].log_data[0].min := 1.0, [2150].log_data[0].max := 1.0, [2150].log_data[0].total := 300.0, [2150].log_data[0].time := 300.0, [2150].log_data[0].minminute := 40, [2150].log_data[0].maxminute := 40, [2150].log_data[0].valid := 1, [2150].log_data[1].valid := 1, [2150].log_data[2].valid := 1, [2150].log_data[3].valid := 1, [2150].log_data[4].valid := 1, [2150].time.Year := 2022, [2150].time.Month := 5, [2150].time.Day := 1, [2150].time.Hour := 8, [2150].time.Minute := 44, [2150].time.Second := 59, [2150].time.DST_ON := 1, [2151].log_data[0].min := 1.0, [2151].log_data[0].max := 1.0, [2151].log_data[0].total := 300.0, [2151].log_data[0].time := 300.0, [2151].log_data[0].minminute := 45, [2151].log_data[0].maxminute := 45, [2151].log_data[0].valid := 1, [2151].log_data[1].valid := 1, [2151].log_data[2].valid := 1, [2151].log_data[3].valid := 1, [2151].log_data[4].valid := 1,
        [2151].time.Year := 2022, [2151].time.Month := 5, [2151].time.Day := 1, [2151].time.Hour := 8, [2151].time.Minute := 49, [2151].time.Second := 59, [2151].time.DST_ON := 1, [2152].log_data[0].min := 1.0, [2152].log_data[0].max := 1.0, [2152].log_data[0].total := 300.0, [2152].log_data[0].time := 300.0, [2152].log_data[0].minminute := 50, [2152].log_data[0].maxminute := 50, [2152].log_data[0].valid := 1, [2152].log_data[1].valid := 1, [2152].log_data[2].valid := 1, [2152].log_data[3].valid := 1, [2152].log_data[4].valid := 1, [2152].time.Year := 2022, [2152].time.Month := 5, [2152].time.Day := 1, [2152].time.Hour := 8, [2152].time.Minute := 54, [2152].time.Second := 59, [2152].time.DST_ON := 1, [2153].log_data[0].min := 1.0, [2153].log_data[0].max := 1.0, [2153].log_data[0].total := 300.0, [2153].log_data[0].time := 300.0, [2153].log_data[0].minminute := 55, [2153].log_data[0].maxminute := 55, [2153].log_data[0].valid := 1, [2153].log_data[1].valid := 1, [2153].log_data[2].valid := 1, [2153].log_data[3].valid := 1, [2153].log_data[4].valid := 1, [2153].time.Year := 2022, [2153].time.Month := 5, [2153].time.Day := 1, [2153].time.Hour := 8, [2153].time.Minute := 59, [2153].time.Second := 59, [2153].time.DST_ON := 1, [2154].log_data[0].min := 1.0, [2154].log_data[0].max := 1.0, [2154].log_data[0].total := 300.0, [2154].log_data[0].time := 300.0, [2154].log_data[0].valid := 1, [2154].log_data[1].valid := 1, [2154].log_data[2].valid := 1, [2154].log_data[3].valid := 1, [2154].log_data[4].valid := 1, [2154].time.Year := 2022, [2154].time.Month := 5, [2154].time.Day := 1, [2154].time.Hour := 9, [2154].time.Minute := 4, [2154].time.Second := 59, [2154].time.DST_ON := 1, [2155].log_data[0].min := 1.0,
        [2155].log_data[0].max := 1.0, [2155].log_data[0].total := 300.0, [2155].log_data[0].time := 300.0, [2155].log_data[0].minminute := 5, [2155].log_data[0].maxminute := 5, [2155].log_data[0].valid := 1, [2155].log_data[1].valid := 1, [2155].log_data[2].valid := 1, [2155].log_data[3].valid := 1, [2155].log_data[4].valid := 1, [2155].time.Year := 2022, [2155].time.Month := 5, [2155].time.Day := 1, [2155].time.Hour := 9, [2155].time.Minute := 9, [2155].time.Second := 59, [2155].time.DST_ON := 1, [2156].log_data[0].min := 1.0, [2156].log_data[0].max := 1.0, [2156].log_data[0].total := 300.0, [2156].log_data[0].time := 300.0, [2156].log_data[0].minminute := 10, [2156].log_data[0].maxminute := 10, [2156].log_data[0].valid := 1, [2156].log_data[1].valid := 1, [2156].log_data[2].valid := 1, [2156].log_data[3].valid := 1, [2156].log_data[4].valid := 1, [2156].time.Year := 2022, [2156].time.Month := 5, [2156].time.Day := 1, [2156].time.Hour := 9, [2156].time.Minute := 14, [2156].time.Second := 59, [2156].time.DST_ON := 1, [2157].log_data[0].min := 1.0, [2157].log_data[0].max := 1.0, [2157].log_data[0].total := 300.0, [2157].log_data[0].time := 300.0, [2157].log_data[0].minminute := 15, [2157].log_data[0].maxminute := 15, [2157].log_data[0].valid := 1, [2157].log_data[1].valid := 1, [2157].log_data[2].valid := 1, [2157].log_data[3].valid := 1, [2157].log_data[4].valid := 1, [2157].time.Year := 2022, [2157].time.Month := 5, [2157].time.Day := 1, [2157].time.Hour := 9, [2157].time.Minute := 19, [2157].time.Second := 59, [2157].time.DST_ON := 1, [2158].log_data[0].min := 1.0, [2158].log_data[0].max := 1.0, [2158].log_data[0].total := 300.0, [2158].log_data[0].time := 300.0, [2158].log_data[0].minminute := 20, [2158].log_data[0].maxminute := 20, [2158].log_data[0].valid := 1,
        [2158].log_data[1].valid := 1, [2158].log_data[2].valid := 1, [2158].log_data[3].valid := 1, [2158].log_data[4].valid := 1, [2158].time.Year := 2022, [2158].time.Month := 5, [2158].time.Day := 1, [2158].time.Hour := 9, [2158].time.Minute := 24, [2158].time.Second := 59, [2158].time.DST_ON := 1, [2159].log_data[0].min := 1.0, [2159].log_data[0].max := 1.0, [2159].log_data[0].total := 300.0, [2159].log_data[0].time := 300.0, [2159].log_data[0].minminute := 25, [2159].log_data[0].maxminute := 25, [2159].log_data[0].valid := 1, [2159].log_data[1].valid := 1, [2159].log_data[2].valid := 1, [2159].log_data[3].valid := 1, [2159].log_data[4].valid := 1, [2159].time.Year := 2022, [2159].time.Month := 5, [2159].time.Day := 1, [2159].time.Hour := 9, [2159].time.Minute := 29, [2159].time.Second := 59, [2159].time.DST_ON := 1, [2160].log_data[0].min := 1.0, [2160].log_data[0].max := 1.0, [2160].log_data[0].total := 300.0, [2160].log_data[0].time := 300.0, [2160].log_data[0].minminute := 30, [2160].log_data[0].maxminute := 30, [2160].log_data[0].valid := 1, [2160].log_data[1].valid := 1, [2160].log_data[2].valid := 1, [2160].log_data[3].valid := 1, [2160].log_data[4].valid := 1, [2160].time.Year := 2022, [2160].time.Month := 5, [2160].time.Day := 1, [2160].time.Hour := 9, [2160].time.Minute := 34, [2160].time.Second := 59, [2160].time.DST_ON := 1, [2161].log_data[0].min := 1.0, [2161].log_data[0].max := 1.0, [2161].log_data[0].total := 300.0, [2161].log_data[0].time := 300.0, [2161].log_data[0].minminute := 35, [2161].log_data[0].maxminute := 35, [2161].log_data[0].valid := 1, [2161].log_data[1].valid := 1, [2161].log_data[2].valid := 1, [2161].log_data[3].valid := 1, [2161].log_data[4].valid := 1, [2161].time.Year := 2022, [2161].time.Month := 5,
        [2161].time.Day := 1, [2161].time.Hour := 9, [2161].time.Minute := 39, [2161].time.Second := 59, [2161].time.DST_ON := 1, [2162].log_data[0].min := 1.0, [2162].log_data[0].max := 1.0, [2162].log_data[0].total := 300.0, [2162].log_data[0].time := 300.0, [2162].log_data[0].minminute := 40, [2162].log_data[0].maxminute := 40, [2162].log_data[0].valid := 1, [2162].log_data[1].valid := 1, [2162].log_data[2].valid := 1, [2162].log_data[3].valid := 1, [2162].log_data[4].valid := 1, [2162].time.Year := 2022, [2162].time.Month := 5, [2162].time.Day := 1, [2162].time.Hour := 9, [2162].time.Minute := 44, [2162].time.Second := 59, [2162].time.DST_ON := 1, [2163].log_data[0].min := 1.0, [2163].log_data[0].max := 1.0, [2163].log_data[0].total := 300.0, [2163].log_data[0].time := 300.0, [2163].log_data[0].minminute := 45, [2163].log_data[0].maxminute := 45, [2163].log_data[0].valid := 1, [2163].log_data[1].valid := 1, [2163].log_data[2].valid := 1, [2163].log_data[3].valid := 1, [2163].log_data[4].valid := 1, [2163].time.Year := 2022, [2163].time.Month := 5, [2163].time.Day := 1, [2163].time.Hour := 9, [2163].time.Minute := 49, [2163].time.Second := 59, [2163].time.DST_ON := 1, [2164].log_data[0].min := 1.0, [2164].log_data[0].max := 1.0, [2164].log_data[0].total := 300.0, [2164].log_data[0].time := 300.0, [2164].log_data[0].minminute := 50, [2164].log_data[0].maxminute := 50, [2164].log_data[0].valid := 1, [2164].log_data[1].valid := 1, [2164].log_data[2].valid := 1, [2164].log_data[3].valid := 1, [2164].log_data[4].valid := 1, [2164].time.Year := 2022, [2164].time.Month := 5, [2164].time.Day := 1, [2164].time.Hour := 9, [2164].time.Minute := 54, [2164].time.Second := 59, [2164].time.DST_ON := 1, [2165].log_data[0].min := 1.0,
        [2165].log_data[0].max := 1.0, [2165].log_data[0].total := 300.0, [2165].log_data[0].time := 300.0, [2165].log_data[0].minminute := 55, [2165].log_data[0].maxminute := 55, [2165].log_data[0].valid := 1, [2165].log_data[1].valid := 1, [2165].log_data[2].valid := 1, [2165].log_data[3].valid := 1, [2165].log_data[4].valid := 1, [2165].time.Year := 2022, [2165].time.Month := 5, [2165].time.Day := 1, [2165].time.Hour := 9, [2165].time.Minute := 59, [2165].time.Second := 59, [2165].time.DST_ON := 1, [2166].log_data[0].min := 1.0, [2166].log_data[0].max := 1.0, [2166].log_data[0].total := 300.0, [2166].log_data[0].time := 300.0, [2166].log_data[0].valid := 1, [2166].log_data[1].valid := 1, [2166].log_data[2].valid := 1, [2166].log_data[3].valid := 1, [2166].log_data[4].valid := 1, [2166].time.Year := 2022, [2166].time.Month := 5, [2166].time.Day := 1, [2166].time.Hour := 10, [2166].time.Minute := 4, [2166].time.Second := 59, [2166].time.DST_ON := 1, [2167].log_data[0].min := 1.0, [2167].log_data[0].max := 1.0, [2167].log_data[0].total := 300.0, [2167].log_data[0].time := 300.0, [2167].log_data[0].minminute := 5, [2167].log_data[0].maxminute := 5, [2167].log_data[0].valid := 1, [2167].log_data[1].valid := 1, [2167].log_data[2].valid := 1, [2167].log_data[3].valid := 1, [2167].log_data[4].valid := 1, [2167].time.Year := 2022, [2167].time.Month := 5, [2167].time.Day := 1, [2167].time.Hour := 10, [2167].time.Minute := 9, [2167].time.Second := 59, [2167].time.DST_ON := 1, [2168].log_data[0].min := 1.0, [2168].log_data[0].max := 1.0, [2168].log_data[0].total := 300.0, [2168].log_data[0].time := 300.0, [2168].log_data[0].minminute := 10, [2168].log_data[0].maxminute := 10, [2168].log_data[0].valid := 1, [2168].log_data[1].valid := 1, [2168].log_data[2].valid := 1,
        [2168].log_data[3].valid := 1, [2168].log_data[4].valid := 1, [2168].time.Year := 2022, [2168].time.Month := 5, [2168].time.Day := 1, [2168].time.Hour := 10, [2168].time.Minute := 14, [2168].time.Second := 59, [2168].time.DST_ON := 1, [2169].log_data[0].min := 1.0, [2169].log_data[0].max := 1.0, [2169].log_data[0].total := 300.0, [2169].log_data[0].time := 300.0, [2169].log_data[0].minminute := 15, [2169].log_data[0].maxminute := 15, [2169].log_data[0].valid := 1, [2169].log_data[1].valid := 1, [2169].log_data[2].valid := 1, [2169].log_data[3].valid := 1, [2169].log_data[4].valid := 1, [2169].time.Year := 2022, [2169].time.Month := 5, [2169].time.Day := 1, [2169].time.Hour := 10, [2169].time.Minute := 19, [2169].time.Second := 59, [2169].time.DST_ON := 1, [2170].log_data[0].min := 1.0, [2170].log_data[0].max := 1.0, [2170].log_data[0].total := 300.0, [2170].log_data[0].time := 300.0, [2170].log_data[0].minminute := 20, [2170].log_data[0].maxminute := 20, [2170].log_data[0].valid := 1, [2170].log_data[1].valid := 1, [2170].log_data[2].valid := 1, [2170].log_data[3].valid := 1, [2170].log_data[4].valid := 1, [2170].time.Year := 2022, [2170].time.Month := 5, [2170].time.Day := 1, [2170].time.Hour := 10, [2170].time.Minute := 24, [2170].time.Second := 59, [2170].time.DST_ON := 1, [2171].log_data[0].min := 1.0, [2171].log_data[0].max := 1.0, [2171].log_data[0].total := 300.0, [2171].log_data[0].time := 300.0, [2171].log_data[0].minminute := 25, [2171].log_data[0].maxminute := 25, [2171].log_data[0].valid := 1, [2171].log_data[1].valid := 1, [2171].log_data[2].valid := 1, [2171].log_data[3].valid := 1, [2171].log_data[4].valid := 1, [2171].time.Year := 2022, [2171].time.Month := 5, [2171].time.Day := 1, [2171].time.Hour := 10,
        [2171].time.Minute := 29, [2171].time.Second := 59, [2171].time.DST_ON := 1, [2172].log_data[0].min := 1.0, [2172].log_data[0].max := 1.0, [2172].log_data[0].total := 300.0, [2172].log_data[0].time := 300.0, [2172].log_data[0].minminute := 30, [2172].log_data[0].maxminute := 30, [2172].log_data[0].valid := 1, [2172].log_data[1].valid := 1, [2172].log_data[2].valid := 1, [2172].log_data[3].valid := 1, [2172].log_data[4].valid := 1, [2172].time.Year := 2022, [2172].time.Month := 5, [2172].time.Day := 1, [2172].time.Hour := 10, [2172].time.Minute := 34, [2172].time.Second := 59, [2172].time.DST_ON := 1, [2173].log_data[0].min := 1.0, [2173].log_data[0].max := 1.0, [2173].log_data[0].total := 300.0, [2173].log_data[0].time := 300.0, [2173].log_data[0].minminute := 35, [2173].log_data[0].maxminute := 35, [2173].log_data[0].valid := 1, [2173].log_data[1].valid := 1, [2173].log_data[2].valid := 1, [2173].log_data[3].valid := 1, [2173].log_data[4].valid := 1, [2173].time.Year := 2022, [2173].time.Month := 5, [2173].time.Day := 1, [2173].time.Hour := 10, [2173].time.Minute := 39, [2173].time.Second := 59, [2173].time.DST_ON := 1, [2174].log_data[0].min := 1.0, [2174].log_data[0].max := 1.0, [2174].log_data[0].total := 300.0, [2174].log_data[0].time := 300.0, [2174].log_data[0].minminute := 40, [2174].log_data[0].maxminute := 40, [2174].log_data[0].valid := 1, [2174].log_data[1].valid := 1, [2174].log_data[2].valid := 1, [2174].log_data[3].valid := 1, [2174].log_data[4].valid := 1, [2174].time.Year := 2022, [2174].time.Month := 5, [2174].time.Day := 1, [2174].time.Hour := 10, [2174].time.Minute := 44, [2174].time.Second := 59, [2174].time.DST_ON := 1, [2175].log_data[0].min := 1.0, [2175].log_data[0].max := 1.0, [2175].log_data[0].total := 300.0,
        [2175].log_data[0].time := 300.0, [2175].log_data[0].minminute := 45, [2175].log_data[0].maxminute := 45, [2175].log_data[0].valid := 1, [2175].log_data[1].valid := 1, [2175].log_data[2].valid := 1, [2175].log_data[3].valid := 1, [2175].log_data[4].valid := 1, [2175].time.Year := 2022, [2175].time.Month := 5, [2175].time.Day := 1, [2175].time.Hour := 10, [2175].time.Minute := 49, [2175].time.Second := 59, [2175].time.DST_ON := 1, [2176].log_data[0].min := 1.0, [2176].log_data[0].max := 1.0, [2176].log_data[0].total := 300.0, [2176].log_data[0].time := 300.0, [2176].log_data[0].minminute := 50, [2176].log_data[0].maxminute := 50, [2176].log_data[0].valid := 1, [2176].log_data[1].valid := 1, [2176].log_data[2].valid := 1, [2176].log_data[3].valid := 1, [2176].log_data[4].valid := 1, [2176].time.Year := 2022, [2176].time.Month := 5, [2176].time.Day := 1, [2176].time.Hour := 10, [2176].time.Minute := 54, [2176].time.Second := 59, [2176].time.DST_ON := 1, [2177].log_data[0].min := 1.0, [2177].log_data[0].max := 1.0, [2177].log_data[0].total := 300.0, [2177].log_data[0].time := 300.0, [2177].log_data[0].minminute := 55, [2177].log_data[0].maxminute := 55, [2177].log_data[0].valid := 1, [2177].log_data[1].valid := 1, [2177].log_data[2].valid := 1, [2177].log_data[3].valid := 1, [2177].log_data[4].valid := 1, [2177].time.Year := 2022, [2177].time.Month := 5, [2177].time.Day := 1, [2177].time.Hour := 10, [2177].time.Minute := 59, [2177].time.Second := 59, [2177].time.DST_ON := 1, [2178].log_data[0].min := 1.0, [2178].log_data[0].max := 1.0, [2178].log_data[0].total := 300.0, [2178].log_data[0].time := 300.0, [2178].log_data[0].valid := 1, [2178].log_data[1].valid := 1, [2178].log_data[2].valid := 1, [2178].log_data[3].valid := 1, [2178].log_data[4].valid := 1,
        [2178].time.Year := 2022, [2178].time.Month := 5, [2178].time.Day := 1, [2178].time.Hour := 11, [2178].time.Minute := 4, [2178].time.Second := 59, [2178].time.DST_ON := 1, [2179].log_data[0].min := 1.0, [2179].log_data[0].max := 1.0, [2179].log_data[0].total := 300.0, [2179].log_data[0].time := 300.0, [2179].log_data[0].minminute := 5, [2179].log_data[0].maxminute := 5, [2179].log_data[0].valid := 1, [2179].log_data[1].valid := 1, [2179].log_data[2].valid := 1, [2179].log_data[3].valid := 1, [2179].log_data[4].valid := 1, [2179].time.Year := 2022, [2179].time.Month := 5, [2179].time.Day := 1, [2179].time.Hour := 11, [2179].time.Minute := 9, [2179].time.Second := 59, [2179].time.DST_ON := 1, [2180].log_data[0].min := 1.0, [2180].log_data[0].max := 1.0, [2180].log_data[0].total := 300.0, [2180].log_data[0].time := 300.0, [2180].log_data[0].minminute := 10, [2180].log_data[0].maxminute := 10, [2180].log_data[0].valid := 1, [2180].log_data[1].valid := 1, [2180].log_data[2].valid := 1, [2180].log_data[3].valid := 1, [2180].log_data[4].valid := 1, [2180].time.Year := 2022, [2180].time.Month := 5, [2180].time.Day := 1, [2180].time.Hour := 11, [2180].time.Minute := 14, [2180].time.Second := 59, [2180].time.DST_ON := 1, [2181].log_data[0].min := 1.0, [2181].log_data[0].max := 1.0, [2181].log_data[0].total := 300.0, [2181].log_data[0].time := 300.0, [2181].log_data[0].minminute := 15, [2181].log_data[0].maxminute := 15, [2181].log_data[0].valid := 1, [2181].log_data[1].valid := 1, [2181].log_data[2].valid := 1, [2181].log_data[3].valid := 1, [2181].log_data[4].valid := 1, [2181].time.Year := 2022, [2181].time.Month := 5, [2181].time.Day := 1, [2181].time.Hour := 11, [2181].time.Minute := 19, [2181].time.Second := 59,
        [2181].time.DST_ON := 1, [2182].log_data[0].min := 1.0, [2182].log_data[0].max := 1.0, [2182].log_data[0].total := 300.0, [2182].log_data[0].time := 300.0, [2182].log_data[0].minminute := 20, [2182].log_data[0].maxminute := 20, [2182].log_data[0].valid := 1, [2182].log_data[1].valid := 1, [2182].log_data[2].valid := 1, [2182].log_data[3].valid := 1, [2182].log_data[4].valid := 1, [2182].time.Year := 2022, [2182].time.Month := 5, [2182].time.Day := 1, [2182].time.Hour := 11, [2182].time.Minute := 24, [2182].time.Second := 59, [2182].time.DST_ON := 1, [2183].log_data[0].min := 1.0, [2183].log_data[0].max := 1.0, [2183].log_data[0].total := 300.0, [2183].log_data[0].time := 300.0, [2183].log_data[0].minminute := 25, [2183].log_data[0].maxminute := 25, [2183].log_data[0].valid := 1, [2183].log_data[1].valid := 1, [2183].log_data[2].valid := 1, [2183].log_data[3].valid := 1, [2183].log_data[4].valid := 1, [2183].time.Year := 2022, [2183].time.Month := 5, [2183].time.Day := 1, [2183].time.Hour := 11, [2183].time.Minute := 29, [2183].time.Second := 59, [2183].time.DST_ON := 1, [2184].log_data[0].min := 1.0, [2184].log_data[0].max := 1.0, [2184].log_data[0].total := 300.0, [2184].log_data[0].time := 300.0, [2184].log_data[0].minminute := 30, [2184].log_data[0].maxminute := 30, [2184].log_data[0].valid := 1, [2184].log_data[1].valid := 1, [2184].log_data[2].valid := 1, [2184].log_data[3].valid := 1, [2184].log_data[4].valid := 1, [2184].time.Year := 2022, [2184].time.Month := 5, [2184].time.Day := 1, [2184].time.Hour := 11, [2184].time.Minute := 34, [2184].time.Second := 59, [2184].time.DST_ON := 1, [2185].log_data[0].min := 1.0, [2185].log_data[0].max := 1.0, [2185].log_data[0].total := 300.0, [2185].log_data[0].time := 300.0, [2185].log_data[0].minminute := 35,
